Omron Sysmac Studio project Cobot_Test_200521 (Sysmac Studio 1.40.0.64008, StandardProject)

# Controller new_Controller_0: NX102-9020 version 1.34
Units and slaves: Unit 1 : NX-PF0730 (N2); Unit 2 : NX-AD3203 (N3); Unit 3 : NX-ID5442 (N4); Unit 4 : NX-OC4633 (N1); Unit 5 : NX-OC4633 (N7)
Task PrimaryTask (priority 4, period or condition 2000): Main, TM_Movements_Connection, TM_Movements, CobotModbusComms
Library TM_Commands 1.2.1 (contents left out)
Library TMmodbus Lib FW1.80 FB3.0.03 3.0.03 (contents left out)

TYPE PointStruct : STRUCT
    PosX : REAL;
    PosY : REAL;
    PosZ : REAL;
    PosRx : REAL;
    PosRy : REAL;
    PosRz : REAL;
END_STRUCT END_TYPE
TYPE PointStruct_STR : STRUCT
    PosX : STRING[10];
    PosY : STRING[10];
    PosZ : STRING[10];
    PosRx : STRING[10];
    PosRy : STRING[10];
    PosRz : STRING[10];
END_STRUCT END_TYPE
TYPE RobPosDK : STRUCT  (* TM12 move cmd from RoboDK *)
    MovType : STRING[15];  (* Move Type (PTP,Line,Circle) *)
    RobPosX : REAL;  (* X axis coordinates *)
    RobPosY : REAL;  (* Y axis coordinates *)
    RobPosZ : REAL;  (* Z axis coordinates *)
    RobPosRx : REAL;  (* Rotational X axis coordinates *)
    RobPosRy : REAL;  (* Rotational Y axis coordinates *)
    RobPosRz : REAL;  (* Rotational Z axis coordinates *)
    VarIO : STRING[20];
END_STRUCT END_TYPE
TYPE JobStruct : STRUCT
    JobID : INT;
    PartID : STRING[50];
    Qty : INT;
    EstTime : STRING[50];
    StartTimeDate : STRING[50];
    JobType : STRING[50];
    TimeAdded : DATE_AND_TIME;
END_STRUCT END_TYPE

VAR_GLOBAL RETAIN
    StartCommunications : BOOL;  (* published *)
END_VAR
VAR_GLOBAL
    MBerror : WORD;  (* published *)
    RobotCoordinates : TMmodbus\sRobotCoordinate;  (* published *)
    TouchCoordinates : TMmodbus\sRobotCoordinateTouch;  (* published *)
    RobotStatus : TMmodbus\sRobotStatus;  (* published *)
    RobotVitals : TMmodbus\sRobotVitals;  (* published *)
    Config : TMmodbus\sConfiguration;  (* published *)
    RobotJointTorques : TMmodbus\sRobotJointTorque;  (* published *)
    RobotTCPLive : TMmodbus\sRobotTCPLive;  (* published *)
    CurrentProjectName : string[200];  (* published *)
    NewProjectName : string[200];  (* published *)
    CommsRoundRobin : REAL;  (* published *)
    TCPerror : WORD;  (* published *)
    RobotControlBoxInfo : TMmodbus\sRobotControllerData;  (* published *)
    Buttons : TMmodbus\sRobotStickButtons;  (* published *)
    RobotIO : TMmodbus\sRobotIO;  (* published *)
    RobotSafetySettings : TMmodbus\sRobotSafety;  (* published *)
    RealsToRobot : ARRAY[0..49] OF real;  (* published *)
    FloatsFromRobot : ARRAY[0..49] OF real;  (* published *)
    BoolsToRobot : ARRAY[0..63] OF BOOL;  (* published *)
    Int16sFromRobot : ARRAY[0..49] OF INT;  (* published *)
    BoolsFromRobot : ARRAY[0..63] OF BOOL;  (* published *)
    IntsToRobot : ARRAY[0..49] OF INT;  (* published *)
    CommunicationsStatus : _eCONNECTION_STATE;  (* published *)
    CommunicationsBusy : BOOL;  (* published *)
    TCPerrorOriginator : TMModbus\eFunctionBlockError;  (* published *)
    RetryCounter : UINT;  (* published *)
    Stitching_Status : DINT;  (* published *)
    Stitching_Speed : REAL;  (* published *)
    Robot_Status : DINT;  (* published *)
    RobPos_X : DINT;  (* published *)
    RobPos_Y : DINT;  (* published *)
    RobPos_Z : DINT;  (* published *)
    Relay_Output : BYTE;  (* at IOBus://unit#4/Output Bit 8 bits; published *)
    Relay_Output1 : BOOL;  (* at IOBus://unit#4/Output Bit 8 bits/Output Bit 00; published *)
    Relay_Output2 : BOOL;  (* at IOBus://unit#4/Output Bit 8 bits/Output Bit 01; published *)
    Relay_Output3 : BOOL;  (* at IOBus://unit#4/Output Bit 8 bits/Output Bit 02; published *)
    Relay_Output4 : BOOL;  (* at IOBus://unit#4/Output Bit 8 bits/Output Bit 03; published *)
    Run_Stiching : BOOL;  (* published *)
    StartProgram : BOOL;  (* published *)
    CableConnected : BOOL;  (* published *)
    MTCP_Connect_TCP_Socket : _sSOCKET;  (* published *)
    MTCP_Connect_Connected : BOOL;
    ListenNode_Connect_Connected : BOOL;
    ListenNode_Connect_TCP_Socket : _sSOCKET;
    TaskTimeFB : REAL;
    Speed : REAL;  (* published *)
    TM_ReadPosition_X : REAL;
    TM_ReadPosition_Y : REAL;
    TM_ReadPosition_Z : REAL;  (* published *)
    Register : ARRAY[0..1023] OF WORD;
    TM_MovCmd_Command : STRING[256];
    Stitching_InManual : BOOL;
    Vision_IN : ARRAY[0..495] OF BYTE;  (* network input *)
    Vision_OUT : ARRAY[0..495] OF BYTE;  (* network output *)
    Part_Orientation_DINT : DINT;
    Part_Dist_X : DINT;
    Part_Dist_Y : DINT;
    Vision_Result_OK : DINT;  (* published *)
    Part_Orientation_REAL : REAL;
    Rz_Attach : REAL;
    RZ_Attach_String : STRING[256] := '';
    X_Attach_String : String[10];
    Y_Attach_String : STRING[10];
END_VAR
VAR_GLOBAL RETAIN
    AttachPoint : PointStruct;
END_VAR
VAR_GLOBAL
    AttachPoint_STR : PointStruct_STR;
    Z_Attach_String : string[10];
    Rx_Attach_String : string[10];
    Ry_Attach_String : string[10];
    Attach : STRING[256];
    RobPosTM : ARRAY[0..100] OF RobPosDK;
    CSVstrings : ARRAY[0..100] OF STRING[100];
    Position_STR : ARRAY[0..100] OF PointStruct_STR;
    Position1 : STRING[256];
    Position : ARRAY[0..100] OF STRING[100];
    MovType : ARRAY[0..100] OF STRING[100];
    RoboDKLoad : BOOL;  (* published *)
    FileName : STRING[100];  (* published *)
    ProgramToLoad : STRING[100];
    Index_STR : DINT;
    AI_CH1 : INT;  (* at IOBus://unit#2/Ch1 Analog Input Value; published *)
    AI_CH2 : INT;  (* at IOBus://unit#2/Ch2 Analog Input Value; published *)
    AI_CH3 : INT;  (* at IOBus://unit#2/Ch3 Analog Input Value; published *)
    AI_CH4 : INT;  (* at IOBus://unit#2/Ch4 Analog Input Value; published *)
    N4_Input_Bit_00 : BOOL;  (* at IOBus://unit#3/Input Bit 16 bits/Input Bit 00 *)
    N4_Input_Bit_01 : BOOL;  (* at IOBus://unit#3/Input Bit 16 bits/Input Bit 01 *)
    N4_Input_Bit_02 : BOOL;  (* at IOBus://unit#3/Input Bit 16 bits/Input Bit 02 *)
    N4_Input_Bit_03 : BOOL;  (* at IOBus://unit#3/Input Bit 16 bits/Input Bit 03 *)
    N4_Input_Bit_04 : BOOL;  (* at IOBus://unit#3/Input Bit 16 bits/Input Bit 04 *)
    N4_Input_Bit_05 : BOOL;  (* at IOBus://unit#3/Input Bit 16 bits/Input Bit 05 *)
    DistanceSensor : REAL;
    Relay_Output5 : BOOL;  (* at IOBus://unit#4/Output Bit 8 bits/Output Bit 04 *)
    Relay_Output6 : BOOL;  (* at IOBus://unit#4/Output Bit 8 bits/Output Bit 05 *)
    Relay_Output7 : BOOL;  (* at IOBus://unit#4/Output Bit 8 bits/Output Bit 06 *)
    Relay_Output8 : BOOL;  (* at IOBus://unit#4/Output Bit 8 bits/Output Bit 07 *)
    Bottom_Cyl_IN : BOOL;
    Bottom_Cyl_OUT : BOOL;
    Striker_Plt_DOWN : BOOL;
    Striker_Plt_UP : BOOL;
    Cutter_IN : BOOL;
    Cutter_OUT : BOOL;
    Top_N_Bottom_Cut_D : BOOL;
    Striker_Plate_D : BOOL;
    Vacuum_D : BOOL;
    Main_Cut_D : BOOL;
    Alarms_Int : DINT;  (* published *)
    Rob_Speed : DINT;  (* published *)
    GRAFANA_Counter : INT;  (* published *)
    Taping_Status : DINT;  (* published *)
    Run_Taping : BOOL;
END_VAR
VAR_GLOBAL RETAIN
    Parts_06Hrs : DINT;  (* published *)
    Parts_07Hrs : DINT;  (* published *)
    Parts_08Hrs : DINT;  (* published *)
    Parts_09Hrs : DINT;  (* published *)
    Parts_10Hrs : DINT;  (* published *)
    Parts_11Hrs : DINT;  (* published *)
    Parts_12Hrs : DINT;  (* published *)
    Parts_13Hrs : DINT;  (* published *)
    Parts_14Hrs : DINT;  (* published *)
    Parts_15Hrs : DINT;  (* published *)
    Parts_16Hrs : DINT;  (* published *)
    Parts_17Hrs : DINT;  (* published *)
    Parts_SP : DINT;  (* published *)
END_VAR
VAR_GLOBAL
    Stitching_OEE : DINT;  (* published *)
    Taping_OEE : DINT;  (* published *)
    RobProgIO : ARRAY[0..100] OF STRING[25];
    Run_Stiching_Man : BOOL;  (* published *)
    Stitcher_AutoSpeed : BOOL;
    Proj_Rob_Speed : INT;
    VarIO : ARRAY[0..100] OF STRING[100];
    Relay_Output9 : BOOL;  (* at IOBus://unit#5/Output Bit 8 bits/Output Bit 00 *)
    ERPJob : JobStruct;  (* published *)
    ERPJobWorking : JobStruct;
END_VAR
VAR_GLOBAL CONSTANT
    ERPJobZero : JobStruct;
END_VAR

PROGRAM Main
VAR
    Input1 : BOOL;  (* Enter Variable Commen *)
    Input2 : BOOL;
    Input3 : BOOL;
    Input4 : BOOL;
    RobotPos_Stiching : BOOL;
    xPlaceholder : DINT;
    yPlaceholder : DINT;
    zPlaceholder : DINT;
    placeholder : BOOL;
    Robot_Running : BOOL;
    Rb_Error_Present : BOOL;
    St_Error_Present : BOOL;
    CommunicationsBusy : BOOL;
    StartCommunications : BOOL;
    Start : BOOL;
    def : BOOL;
    testt : BOOL;
    X_Attach : REAL;
    Y_Attach : REAL;
    Part_Dist_X_REAL : REAL;
    Part_Dist_Y_REAL : REAL;
    X_temp : REAL;
    Y_temp : REAL;
    TrigRoboProgramRead : BOOL;
    OpenRoboProgram : FileOpen;
    OpenFileError : BOOL;
    ProgramToOpen : STRING[255];
    Fid : DWORD;
    ReadRoboProgram : FileGets;
    ReadFileError : BOOL;
    Index : DINT;
    CloseRoboProgram : FileClose;
    CloseFileError : BOOL;
    ReadComplete : BOOL;
    OperatingEnd : BOOL;
    Trigger : BOOL;
    RS_Instance : RS;
    tuti : BOOL;
    OpenProgramName : STRING[100];
    x : BOOL;
    i : DINT;
    R_TRIG_instance : R_TRIG;
    Stp : DINT;
    Vis_Error_Present : BOOL;
    Rob_Alarm : BOOL;
    St_Alarm : BOOL;
    Vis_Alarm : BOOL;
    GRAFANA_TON : TON;
    GRAFANA_TON_ET : TIME;
    GRAFANA_CTU : CTU;
    Reset_Counter : BOOL;
    Tp_Error_Present : BOOL;
    Tp_Alarm : BOOL;
    Speed_mms : DINT;
    StepMove : DINT;
    temp : UINT;
    Load : BOOL;
    LoadSchedule : BOOL;
    ScheduleName : STRING[100];
    TrigScheduleRead : BOOL;
    OpenSchedule : FileOpen;
    ReadSchedule : FileGets;
    CloseSchedule : FileClose;
    BackStitch_TON : TON;
    BackStitch_TON_ACC : TIME;
    MoveERPData : BOOL;
    abc : _sTimer;
    timeret : UINT;
    q : BOOL;
    TON12 : TON;
    afd : TIME;
    tesss : BOOL;
    ClearERPData : BOOL;
END_VAR
VAR_EXTERNAL
    Stitching_Status : DINT;
    Stitching_Speed : REAL;
    Robot_Status : DINT;
    Relay_Output : BYTE;
    RobPos_X : DINT;
    RobPos_Y : DINT;
    RobPos_Z : DINT;
    RobotCoordinates : TMmodbus\sRobotCoordinate;
    RobotStatus : TMmodbus\sRobotStatus;
    Run_Stiching : BOOL;
    Speed : REAL;
    Vision_IN : ARRAY[0..495] OF BYTE;
    Part_Orientation_DINT : DINT;
    Part_Dist_X : DINT;
    Part_Dist_Y : DINT;
    Vision_OUT : ARRAY[0..495] OF BYTE;
    Part_Orientation_REAL : REAL;
    Rz_Attach : REAL;
    RZ_Attach_String : STRING[256];
    X_Attach_String : String[10];
    Y_Attach_String : STRING[10];
    AttachPoint : PointStruct;
    Z_Attach_String : string[10];
    RX_Attach_String : string[10];
    RY_Attach_String : string[10];
    AttachPoint_STR : PointStruct_STR;
    Attach : STRING[256];
    Vision_Result_OK : DINT;
END_VAR
VAR_EXTERNAL CONSTANT
    _Card1Ready : BOOL;
END_VAR
VAR_EXTERNAL
    RobPosTM : ARRAY[0..100] OF RobPosDK;
    CSVstrings : ARRAY[0..100] OF STRING[100];
    Position1 : STRING[256];
    Position_STR : ARRAY[0..100] OF PointStruct_STR;
    Position : ARRAY[0..100] OF STRING[100];
    MovType : ARRAY[0..100] OF STRING[100];
    RoboDKLoad : BOOL;
    FileName : STRING[100];
    Index_STR : DINT;
    AI_CH1 : INT;
    DistanceSensor : REAL;
    N4_Input_Bit_00 : BOOL;
    N4_Input_Bit_01 : BOOL;
    N4_Input_Bit_02 : BOOL;
    N4_Input_Bit_03 : BOOL;
    N4_Input_Bit_04 : BOOL;
    N4_Input_Bit_05 : BOOL;
    Relay_Output5 : BOOL;
    Relay_Output6 : BOOL;
    Relay_Output7 : BOOL;
    Bottom_Cyl_IN : BOOL;
    Bottom_Cyl_OUT : BOOL;
    Striker_Plt_DOWN : BOOL;
    Striker_Plt_UP : BOOL;
    Cutter_IN : BOOL;
    Cutter_OUT : BOOL;
    Top_N_Bottom_Cut_D : BOOL;
    Striker_Plate_D : BOOL;
    Vacuum_D : BOOL;
    Relay_Output8 : BOOL;
    Main_Cut_D : BOOL;
    ListenNode_Connect_Connected : BOOL;
    Alarms_Int : DINT;
    RobotTCPLive : TMmodbus\sRobotTCPLive;
    Rob_Speed : DINT;
    GRAFANA_Counter : INT;
    Taping_Status : DINT;
    Run_Taping : BOOL;
    RobProgIO : ARRAY[0..100] OF STRING[25];
    Run_Stiching_Man : BOOL;
    Stitcher_AutoSpeed : BOOL;
    StartProgram : BOOL;
    VarIO : ARRAY[0..100] OF STRING[100];
    Relay_Output9 : BOOL;
    ERPJob : JobStruct;
    ERPJobWorking : JobStruct;
END_VAR
VAR_EXTERNAL CONSTANT
    ERPJobZero : JobStruct;
END_VAR
VAR
    _e1 : R_TRIG;
    _p2 : BOOL;
    _p3 : BOOL;
    _p4 : BOOL;
    _p5 : BOOL;
    _p6 : BOOL;
    _p7 : BOOL;
    _p8 : BOOL;
    _p9 : BOOL;
    _p10 : BOOL;
    _p11 : BOOL;
    _p12 : BOOL;
    _p13 : BOOL;
    _p14 : BOOL;
    _p15 : BOOL;
    _p16 : BOOL;
    _e17 : F_TRIG;
    _e18 : F_TRIG;
    _e19 : R_TRIG;
    _e20 : R_TRIG;
    _e21 : R_TRIG;
    _p22 : BOOL;
    _p23 : BOOL;
    _e24 : R_TRIG;
    _e25 : R_TRIG;
END_VAR

(* Section DataToGrafana: ladder, written here as Structured Text *)

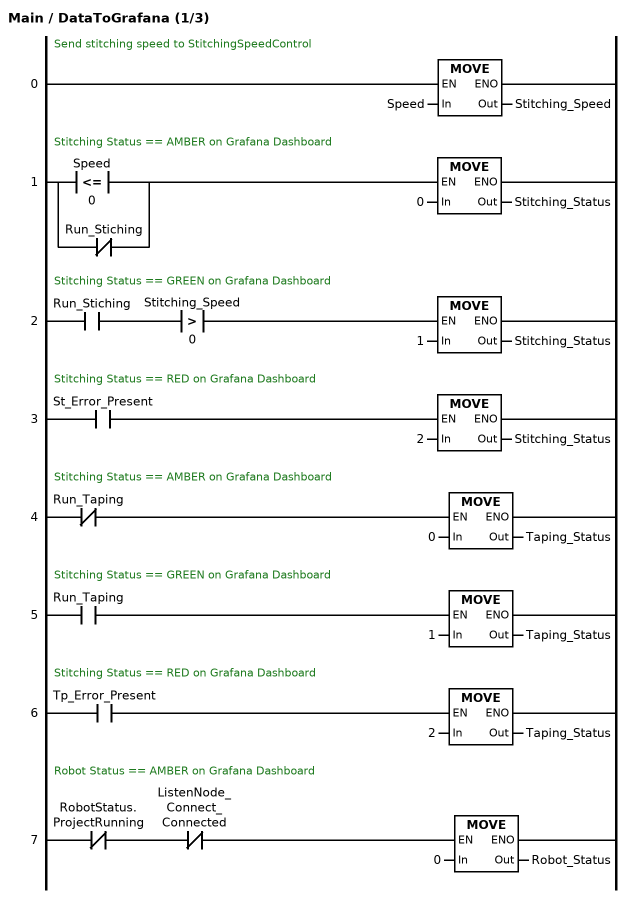
(* Rung 0: Send stitching speed to StitchingSpeedControl *)
Stitching_Speed := Speed;
(* Rung 1: Stitching Status == AMBER on Grafana Dashboard *)
IF (Speed <= 0) OR NOT Run_Stiching THEN Stitching_Status := 0; END_IF;
(* Rung 2: Stitching Status == GREEN on Grafana Dashboard *)
IF Run_Stiching AND (Stitching_Speed > 0) THEN Stitching_Status := 1; END_IF;
(* Rung 3: Stitching Status == RED on Grafana Dashboard *)
IF St_Error_Present THEN Stitching_Status := 2; END_IF;
(* Rung 4: Stitching Status == AMBER on Grafana Dashboard *)
IF NOT Run_Taping THEN Taping_Status := 0; END_IF;
(* Rung 5: Stitching Status == GREEN on Grafana Dashboard *)
IF Run_Taping THEN Taping_Status := 1; END_IF;
(* Rung 6: Stitching Status == RED on Grafana Dashboard *)
IF Tp_Error_Present THEN Taping_Status := 2; END_IF;
(* Rung 7: Robot Status == AMBER on Grafana Dashboard *)
IF NOT RobotStatus.ProjectRunning AND NOT ListenNode_Connect_Connected THEN Robot_Status := 0; END_IF;

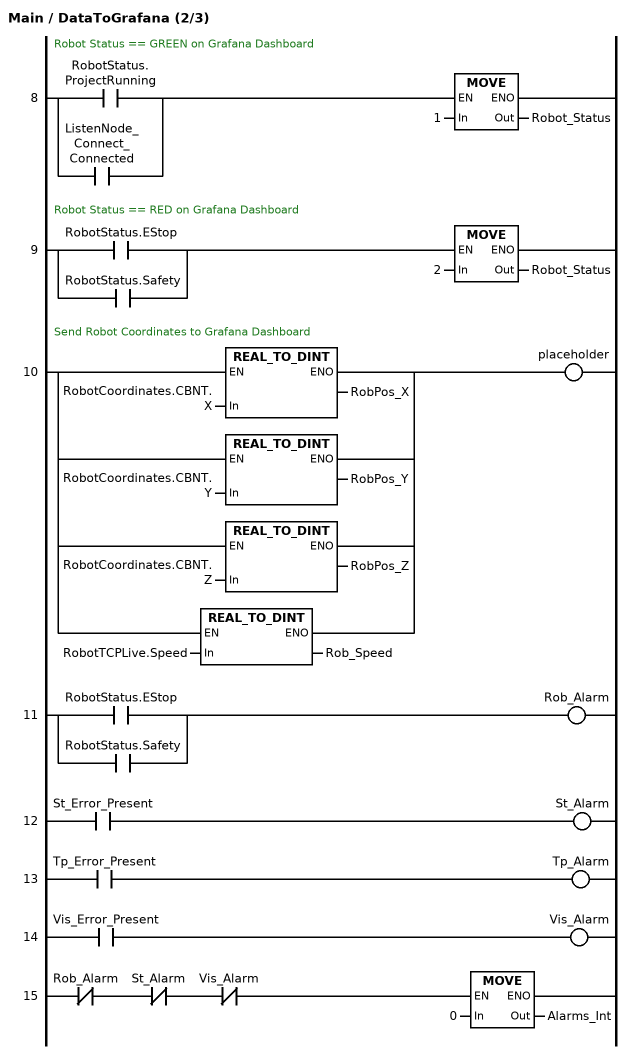
(* Rung 8: Robot Status == GREEN on Grafana Dashboard *)
IF RobotStatus.ProjectRunning OR ListenNode_Connect_Connected THEN Robot_Status := 1; END_IF;
(* Rung 9: Robot Status == RED on Grafana Dashboard *)
IF RobotStatus.EStop OR RobotStatus.Safety THEN Robot_Status := 2; END_IF;
(* Rung 10: Send Robot Coordinates to Grafana Dashboard *)
RobPos_X := REAL_TO_DINT(In := RobotCoordinates.CBNT.X);
RobPos_Y := REAL_TO_DINT(In := RobotCoordinates.CBNT.Y);
RobPos_Z := REAL_TO_DINT(In := RobotCoordinates.CBNT.Z);
Rob_Speed := REAL_TO_DINT(In := RobotTCPLive.Speed);
placeholder := TRUE;
(* Rung 11 *)
Rob_Alarm := RobotStatus.EStop OR RobotStatus.Safety;
(* Rung 12 *)
St_Alarm := St_Error_Present;
(* Rung 13 *)
Tp_Alarm := Tp_Error_Present;
(* Rung 14 *)
Vis_Alarm := Vis_Error_Present;
(* Rung 15 *)
IF NOT Rob_Alarm AND NOT St_Alarm AND NOT Vis_Alarm THEN Alarms_Int := 0; END_IF;

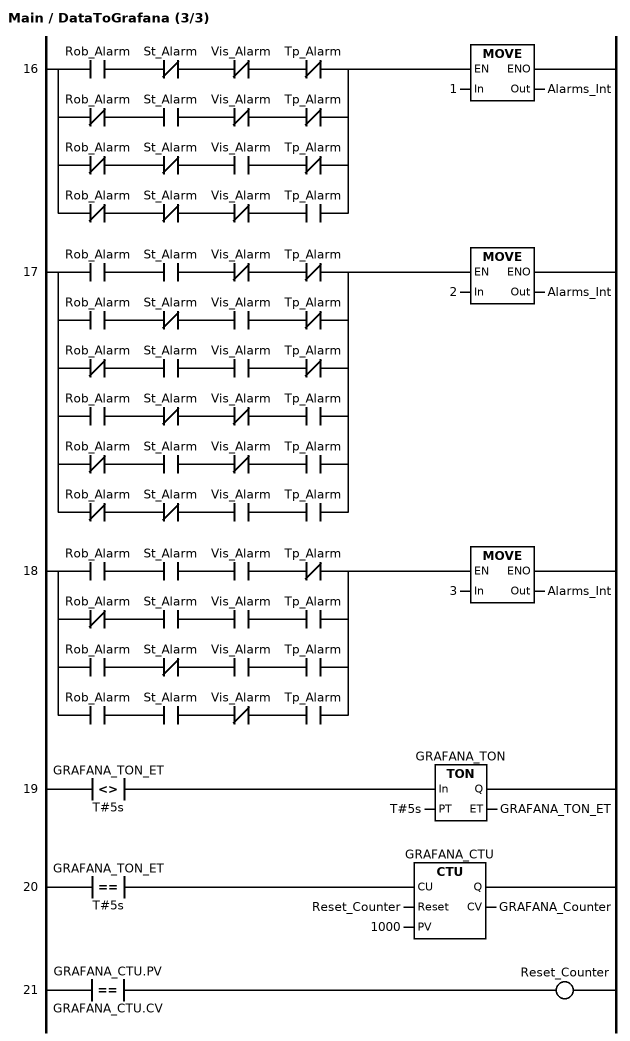
(* Rung 16 *)
IF (Rob_Alarm AND NOT St_Alarm AND NOT Vis_Alarm AND NOT Tp_Alarm) OR (NOT Rob_Alarm AND St_Alarm AND NOT Vis_Alarm AND NOT Tp_Alarm) OR (NOT Rob_Alarm AND NOT St_Alarm AND Vis_Alarm AND NOT Tp_Alarm) OR (NOT Rob_Alarm AND NOT St_Alarm AND NOT Vis_Alarm AND Tp_Alarm) THEN
    Alarms_Int := 1;
END_IF;
(* Rung 17 *)
IF (Rob_Alarm AND St_Alarm AND NOT Vis_Alarm AND NOT Tp_Alarm) OR (Rob_Alarm AND NOT St_Alarm AND Vis_Alarm AND NOT Tp_Alarm) OR (NOT Rob_Alarm AND St_Alarm AND Vis_Alarm AND NOT Tp_Alarm) OR (Rob_Alarm AND NOT St_Alarm AND NOT Vis_Alarm AND Tp_Alarm) OR (NOT Rob_Alarm AND St_Alarm AND NOT Vis_Alarm AND Tp_Alarm) OR (NOT Rob_Alarm AND NOT St_Alarm AND Vis_Alarm AND Tp_Alarm) THEN
    Alarms_Int := 2;
END_IF;
(* Rung 18 *)
IF (Rob_Alarm AND St_Alarm AND Vis_Alarm AND NOT Tp_Alarm) OR (NOT Rob_Alarm AND St_Alarm AND Vis_Alarm AND Tp_Alarm) OR (Rob_Alarm AND NOT St_Alarm AND Vis_Alarm AND Tp_Alarm) OR (Rob_Alarm AND St_Alarm AND NOT Vis_Alarm AND Tp_Alarm) THEN
    Alarms_Int := 3;
END_IF;
(* Rung 19 *)
GRAFANA_TON(In := GRAFANA_TON_ET <> T#5s, PT := T#5s, ET => GRAFANA_TON_ET);
(* Rung 20 *)
_e1(CLK := GRAFANA_TON_ET = T#5s);
GRAFANA_CTU(CU := _e1.Q, Reset := Reset_Counter, PV := 1000, CV => GRAFANA_Counter);
(* Rung 21 *)
Reset_Counter := GRAFANA_CTU.PV = GRAFANA_CTU.CV;

(* Section StichingMachine: ladder, written here as Structured Text *)

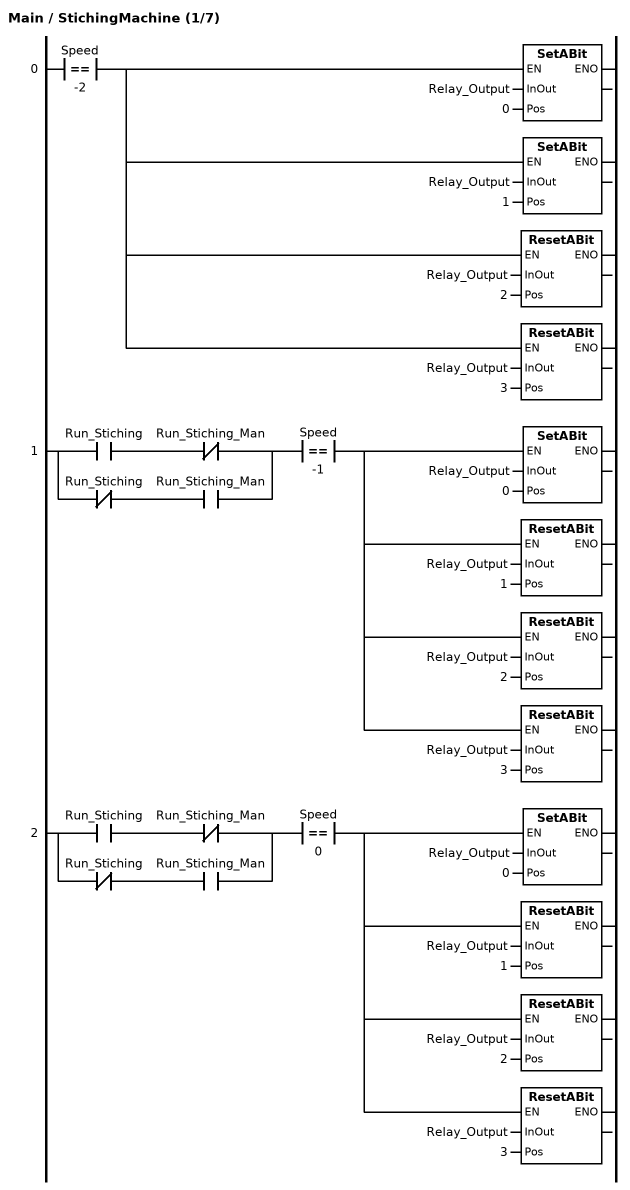
(* Rung 0 *)
IF Speed = -2 THEN
    SetABit(InOut := Relay_Output, Pos := 0);
    SetABit(InOut := Relay_Output, Pos := 1);
    ResetABit(InOut := Relay_Output, Pos := 2);
    ResetABit(InOut := Relay_Output, Pos := 3);
END_IF;
(* Rung 1 *)
_p2 := ((Run_Stiching AND NOT Run_Stiching_Man) OR (NOT Run_Stiching AND Run_Stiching_Man)) AND (Speed = -1);
IF _p2 THEN
    SetABit(InOut := Relay_Output, Pos := 0);
    ResetABit(InOut := Relay_Output, Pos := 1);
    ResetABit(InOut := Relay_Output, Pos := 2);
    ResetABit(InOut := Relay_Output, Pos := 3);
END_IF;
(* Rung 2 *)
_p3 := ((Run_Stiching AND NOT Run_Stiching_Man) OR (NOT Run_Stiching AND Run_Stiching_Man)) AND (Speed = 0);
IF _p3 THEN
    SetABit(InOut := Relay_Output, Pos := 0);
    ResetABit(InOut := Relay_Output, Pos := 1);
    ResetABit(InOut := Relay_Output, Pos := 2);
    ResetABit(InOut := Relay_Output, Pos := 3);
END_IF;

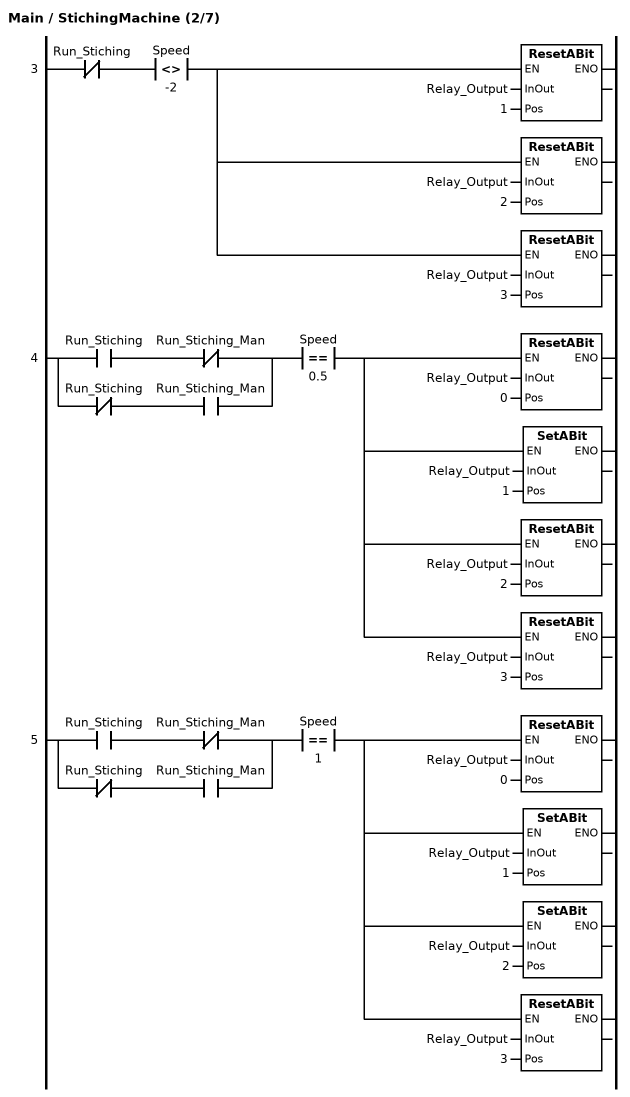
(* Rung 3 *)
IF NOT Run_Stiching AND (Speed <> -2) THEN
    ResetABit(InOut := Relay_Output, Pos := 1);
    ResetABit(InOut := Relay_Output, Pos := 2);
    ResetABit(InOut := Relay_Output, Pos := 3);
END_IF;
(* Rung 4 *)
_p4 := ((Run_Stiching AND NOT Run_Stiching_Man) OR (NOT Run_Stiching AND Run_Stiching_Man)) AND (Speed = 0.5);
IF _p4 THEN
    ResetABit(InOut := Relay_Output, Pos := 0);
    SetABit(InOut := Relay_Output, Pos := 1);
    ResetABit(InOut := Relay_Output, Pos := 2);
    ResetABit(InOut := Relay_Output, Pos := 3);
END_IF;
(* Rung 5 *)
_p5 := ((Run_Stiching AND NOT Run_Stiching_Man) OR (NOT Run_Stiching AND Run_Stiching_Man)) AND (Speed = 1);
IF _p5 THEN
    ResetABit(InOut := Relay_Output, Pos := 0);
    SetABit(InOut := Relay_Output, Pos := 1);
    SetABit(InOut := Relay_Output, Pos := 2);
    ResetABit(InOut := Relay_Output, Pos := 3);
END_IF;

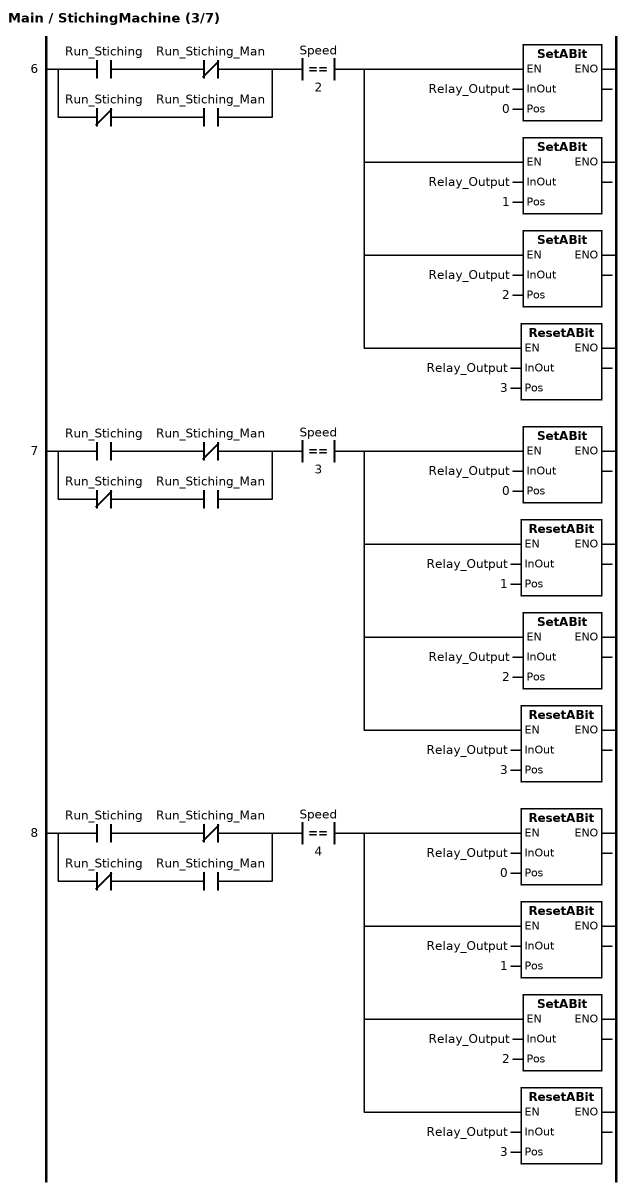
(* Rung 6 *)
_p6 := ((Run_Stiching AND NOT Run_Stiching_Man) OR (NOT Run_Stiching AND Run_Stiching_Man)) AND (Speed = 2);
IF _p6 THEN
    SetABit(InOut := Relay_Output, Pos := 0);
    SetABit(InOut := Relay_Output, Pos := 1);
    SetABit(InOut := Relay_Output, Pos := 2);
    ResetABit(InOut := Relay_Output, Pos := 3);
END_IF;
(* Rung 7 *)
_p7 := ((Run_Stiching AND NOT Run_Stiching_Man) OR (NOT Run_Stiching AND Run_Stiching_Man)) AND (Speed = 3);
IF _p7 THEN
    SetABit(InOut := Relay_Output, Pos := 0);
    ResetABit(InOut := Relay_Output, Pos := 1);
    SetABit(InOut := Relay_Output, Pos := 2);
    ResetABit(InOut := Relay_Output, Pos := 3);
END_IF;
(* Rung 8 *)
_p8 := ((Run_Stiching AND NOT Run_Stiching_Man) OR (NOT Run_Stiching AND Run_Stiching_Man)) AND (Speed = 4);
IF _p8 THEN
    ResetABit(InOut := Relay_Output, Pos := 0);
    ResetABit(InOut := Relay_Output, Pos := 1);
    SetABit(InOut := Relay_Output, Pos := 2);
    ResetABit(InOut := Relay_Output, Pos := 3);
END_IF;

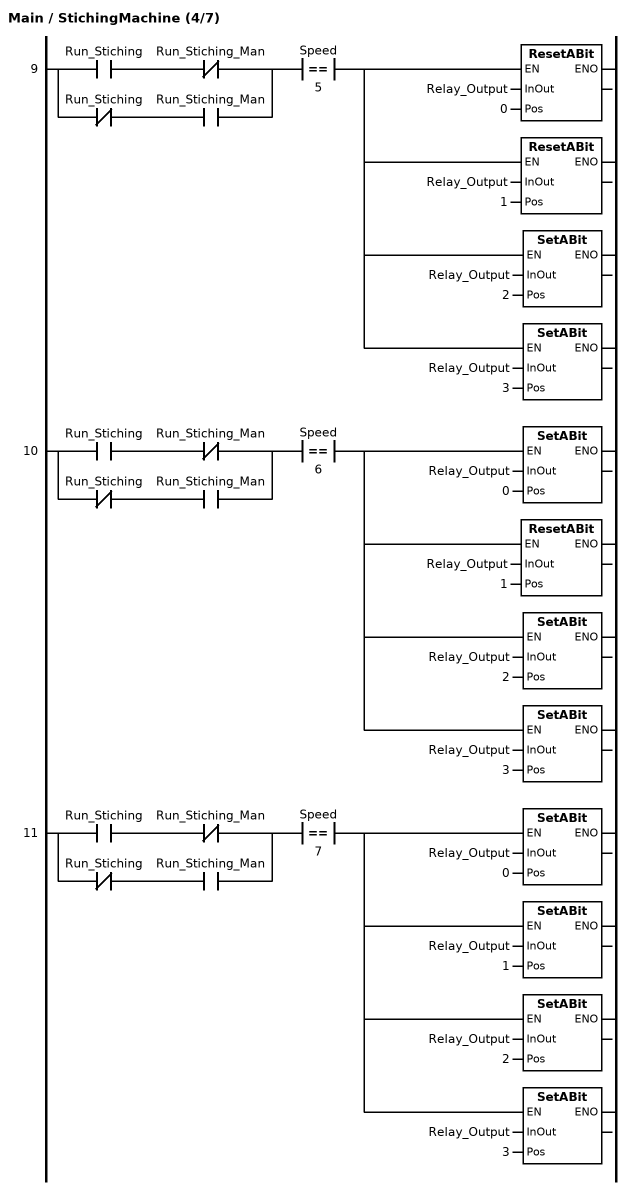
(* Rung 9 *)
_p9 := ((Run_Stiching AND NOT Run_Stiching_Man) OR (NOT Run_Stiching AND Run_Stiching_Man)) AND (Speed = 5);
IF _p9 THEN
    ResetABit(InOut := Relay_Output, Pos := 0);
    ResetABit(InOut := Relay_Output, Pos := 1);
    SetABit(InOut := Relay_Output, Pos := 2);
    SetABit(InOut := Relay_Output, Pos := 3);
END_IF;
(* Rung 10 *)
_p10 := ((Run_Stiching AND NOT Run_Stiching_Man) OR (NOT Run_Stiching AND Run_Stiching_Man)) AND (Speed = 6);
IF _p10 THEN
    SetABit(InOut := Relay_Output, Pos := 0);
    ResetABit(InOut := Relay_Output, Pos := 1);
    SetABit(InOut := Relay_Output, Pos := 2);
    SetABit(InOut := Relay_Output, Pos := 3);
END_IF;
(* Rung 11 *)
_p11 := ((Run_Stiching AND NOT Run_Stiching_Man) OR (NOT Run_Stiching AND Run_Stiching_Man)) AND (Speed = 7);
IF _p11 THEN
    SetABit(InOut := Relay_Output, Pos := 0);
    SetABit(InOut := Relay_Output, Pos := 1);
    SetABit(InOut := Relay_Output, Pos := 2);
    SetABit(InOut := Relay_Output, Pos := 3);
END_IF;

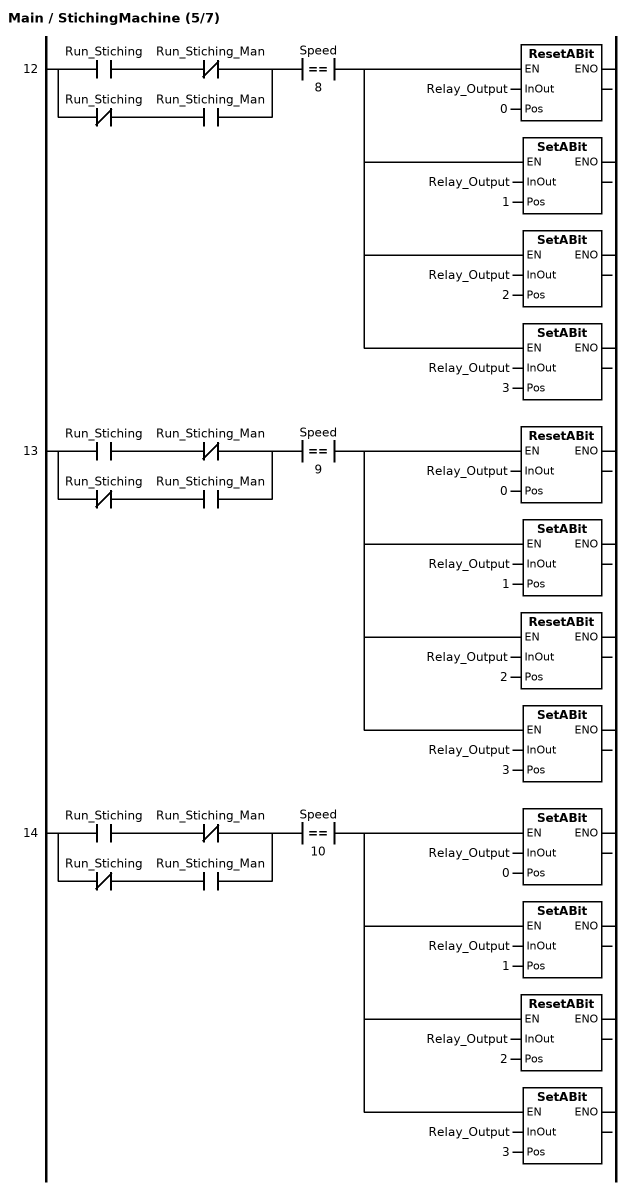
(* Rung 12 *)
_p12 := ((Run_Stiching AND NOT Run_Stiching_Man) OR (NOT Run_Stiching AND Run_Stiching_Man)) AND (Speed = 8);
IF _p12 THEN
    ResetABit(InOut := Relay_Output, Pos := 0);
    SetABit(InOut := Relay_Output, Pos := 1);
    SetABit(InOut := Relay_Output, Pos := 2);
    SetABit(InOut := Relay_Output, Pos := 3);
END_IF;
(* Rung 13 *)
_p13 := ((Run_Stiching AND NOT Run_Stiching_Man) OR (NOT Run_Stiching AND Run_Stiching_Man)) AND (Speed = 9);
IF _p13 THEN
    ResetABit(InOut := Relay_Output, Pos := 0);
    SetABit(InOut := Relay_Output, Pos := 1);
    ResetABit(InOut := Relay_Output, Pos := 2);
    SetABit(InOut := Relay_Output, Pos := 3);
END_IF;
(* Rung 14 *)
_p14 := ((Run_Stiching AND NOT Run_Stiching_Man) OR (NOT Run_Stiching AND Run_Stiching_Man)) AND (Speed = 10);
IF _p14 THEN
    SetABit(InOut := Relay_Output, Pos := 0);
    SetABit(InOut := Relay_Output, Pos := 1);
    ResetABit(InOut := Relay_Output, Pos := 2);
    SetABit(InOut := Relay_Output, Pos := 3);
END_IF;

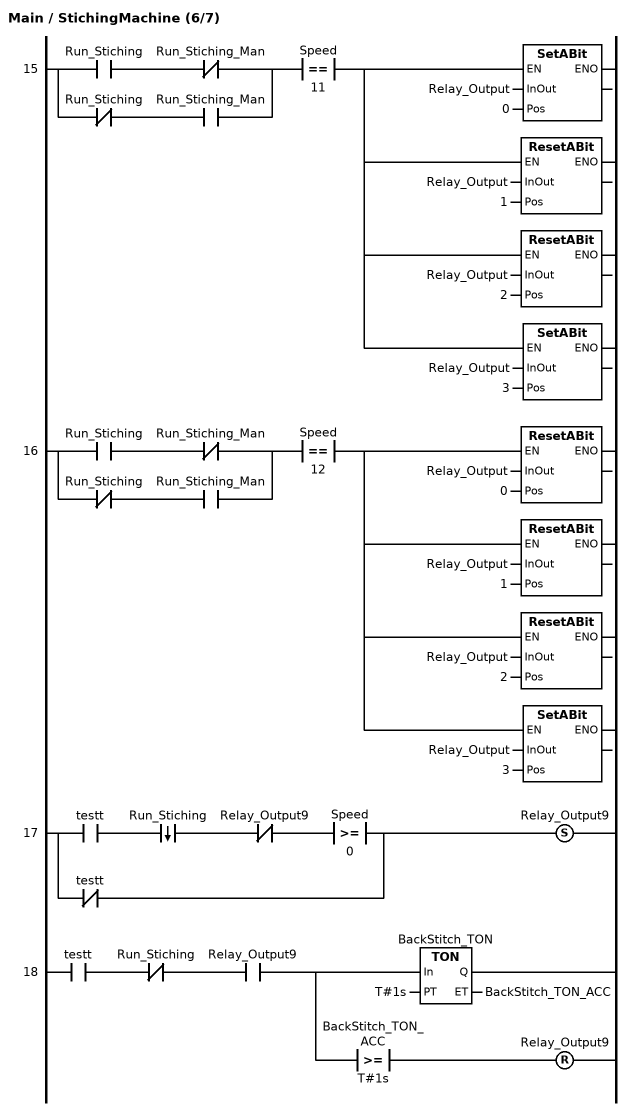
(* Rung 15 *)
_p15 := ((Run_Stiching AND NOT Run_Stiching_Man) OR (NOT Run_Stiching AND Run_Stiching_Man)) AND (Speed = 11);
IF _p15 THEN
    SetABit(InOut := Relay_Output, Pos := 0);
    ResetABit(InOut := Relay_Output, Pos := 1);
    ResetABit(InOut := Relay_Output, Pos := 2);
    SetABit(InOut := Relay_Output, Pos := 3);
END_IF;
(* Rung 16 *)
_p16 := ((Run_Stiching AND NOT Run_Stiching_Man) OR (NOT Run_Stiching AND Run_Stiching_Man)) AND (Speed = 12);
IF _p16 THEN
    ResetABit(InOut := Relay_Output, Pos := 0);
    ResetABit(InOut := Relay_Output, Pos := 1);
    ResetABit(InOut := Relay_Output, Pos := 2);
    SetABit(InOut := Relay_Output, Pos := 3);
END_IF;
(* Rung 17 *)
_e17(CLK := Run_Stiching);
IF (testt AND _e17.Q AND NOT Relay_Output9 AND (Speed >= 0)) OR NOT testt THEN
    Relay_Output9 := TRUE;
END_IF;
(* Rung 18 *)
BackStitch_TON(In := testt AND NOT Run_Stiching AND Relay_Output9, PT := T#1s, ET => BackStitch_TON_ACC);
IF testt AND NOT Run_Stiching AND Relay_Output9 AND (BackStitch_TON_ACC >= T#1s) THEN
    Relay_Output9 := FALSE;
END_IF;

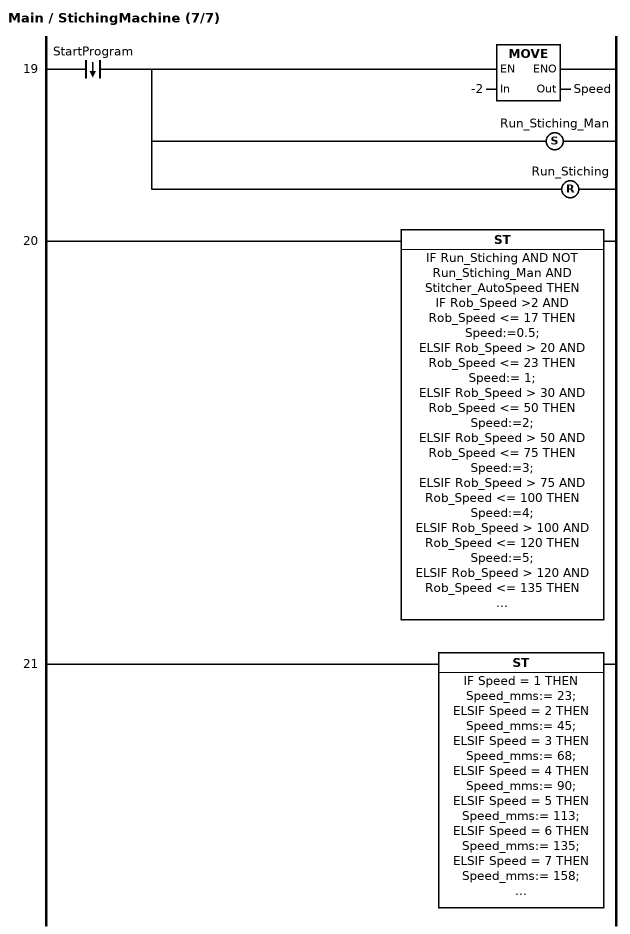
(* Rung 19 *)
_e18(CLK := StartProgram);
IF _e18.Q THEN
    Speed := -2;
    Run_Stiching_Man := TRUE;
    Run_Stiching := FALSE;
END_IF;
(* Rung 20 *)
IF Run_Stiching AND NOT Run_Stiching_Man AND Stitcher_AutoSpeed THEN
	IF Rob_Speed >2 AND Rob_Speed <= 17 THEN
		Speed:=0.5;
	ELSIF Rob_Speed > 20 AND Rob_Speed <= 23 THEN
		Speed:= 1; 
	ELSIF Rob_Speed > 30 AND Rob_Speed <= 50 THEN
		Speed:=2;
	 ELSIF Rob_Speed > 50 AND Rob_Speed <= 75 THEN
		Speed:=3;
	ELSIF Rob_Speed > 75 AND Rob_Speed <= 100 THEN
		Speed:=4;
	ELSIF Rob_Speed > 100 AND Rob_Speed <= 120 THEN
		Speed:=5;
	ELSIF Rob_Speed > 120 AND Rob_Speed <= 135 THEN
		Speed:=6;
	ELSIF Rob_Speed > 135 AND Rob_Speed <= 170 THEN
		Speed:=7;
	ELSIF Rob_Speed > 170 AND Rob_Speed <= 190 THEN
		Speed:=8;
	ELSIF Rob_Speed > 190 AND Rob_Speed <= 210 THEN
		Speed:=9;
	ELSIF Rob_Speed > 210 AND Rob_Speed <= 235 THEN
		Speed:=10;
	ELSIF Rob_Speed > 235 AND Rob_Speed <= 255 THEN
		Speed:=11;
	ELSIF Rob_Speed > 255 AND Rob_Speed <= 270 THEN
		Speed:=12;
	ELSIF Rob_Speed > 270 THEN
		Speed:=12;
	END_IF;
END_IF;
(* Rung 21 *)
IF Speed = 1 THEN
	Speed_mms:= 23;
ELSIF Speed = 2 THEN
	Speed_mms:= 45;
ELSIF Speed = 3 THEN
	Speed_mms:= 68;
ELSIF Speed = 4 THEN
	Speed_mms:= 90;
ELSIF Speed = 5 THEN
	Speed_mms:= 113;
ELSIF Speed = 6 THEN
	Speed_mms:= 135;	
ELSIF Speed = 7 THEN
	Speed_mms:= 158;
ELSIF Speed = 8 THEN
	Speed_mms:= 180;
ELSIF Speed = 9 THEN
	Speed_mms:= 203;
ELSIF Speed = 10 THEN
	Speed_mms:= 225;
ELSIF Speed = 11 THEN
	Speed_mms:= 248;
ELSIF Speed = 12 THEN
	Speed_mms:= 270;
END_IF;

(* Section VisionSystem: ladder, written here as Structured Text *)

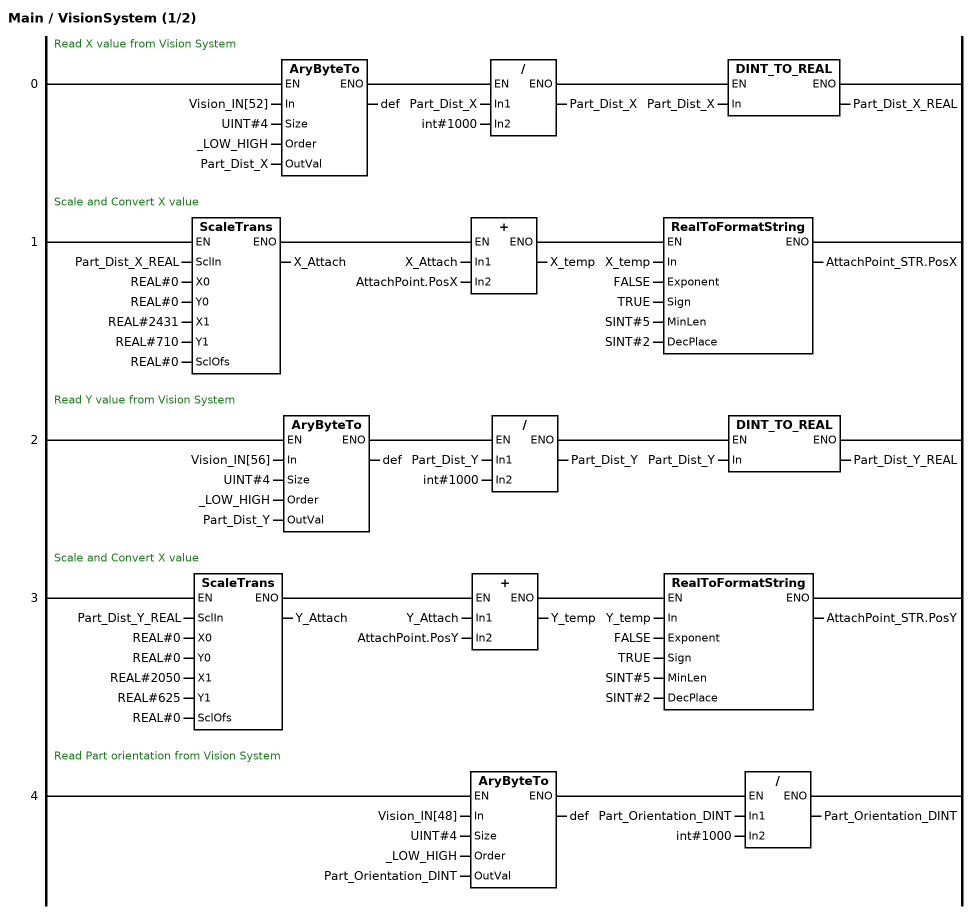
(* Rung 0: Read X value from Vision System *)
def := AryByteTo(In := Vision_IN[52], Size := UINT#4, Order := _LOW_HIGH, OutVal := Part_Dist_X);
Part_Dist_X := Part_Dist_X / int#1000;
Part_Dist_X_REAL := DINT_TO_REAL(In := Part_Dist_X);
(* Rung 1: Scale and Convert X value *)
X_Attach := ScaleTrans(SclIn := Part_Dist_X_REAL, X0 := REAL#0, Y0 := REAL#0, X1 := REAL#2431, Y1 := REAL#710, SclOfs := REAL#0);
X_temp := X_Attach + AttachPoint.PosX;
AttachPoint_STR.PosX := RealToFormatString(In := X_temp, Exponent := FALSE, Sign := TRUE, MinLen := SINT#5, DecPlace := SINT#2);
(* Rung 2: Read Y value from Vision System *)
def := AryByteTo(In := Vision_IN[56], Size := UINT#4, Order := _LOW_HIGH, OutVal := Part_Dist_Y);
Part_Dist_Y := Part_Dist_Y / int#1000;
Part_Dist_Y_REAL := DINT_TO_REAL(In := Part_Dist_Y);
(* Rung 3: Scale and Convert X value *)
Y_Attach := ScaleTrans(SclIn := Part_Dist_Y_REAL, X0 := REAL#0, Y0 := REAL#0, X1 := REAL#2050, Y1 := REAL#625, SclOfs := REAL#0);
Y_temp := Y_Attach + AttachPoint.PosY;
AttachPoint_STR.PosY := RealToFormatString(In := Y_temp, Exponent := FALSE, Sign := TRUE, MinLen := SINT#5, DecPlace := SINT#2);
(* Rung 4: Read Part orientation from Vision System *)
def := AryByteTo(In := Vision_IN[48], Size := UINT#4, Order := _LOW_HIGH, OutVal := Part_Orientation_DINT);
Part_Orientation_DINT := Part_Orientation_DINT / int#1000;

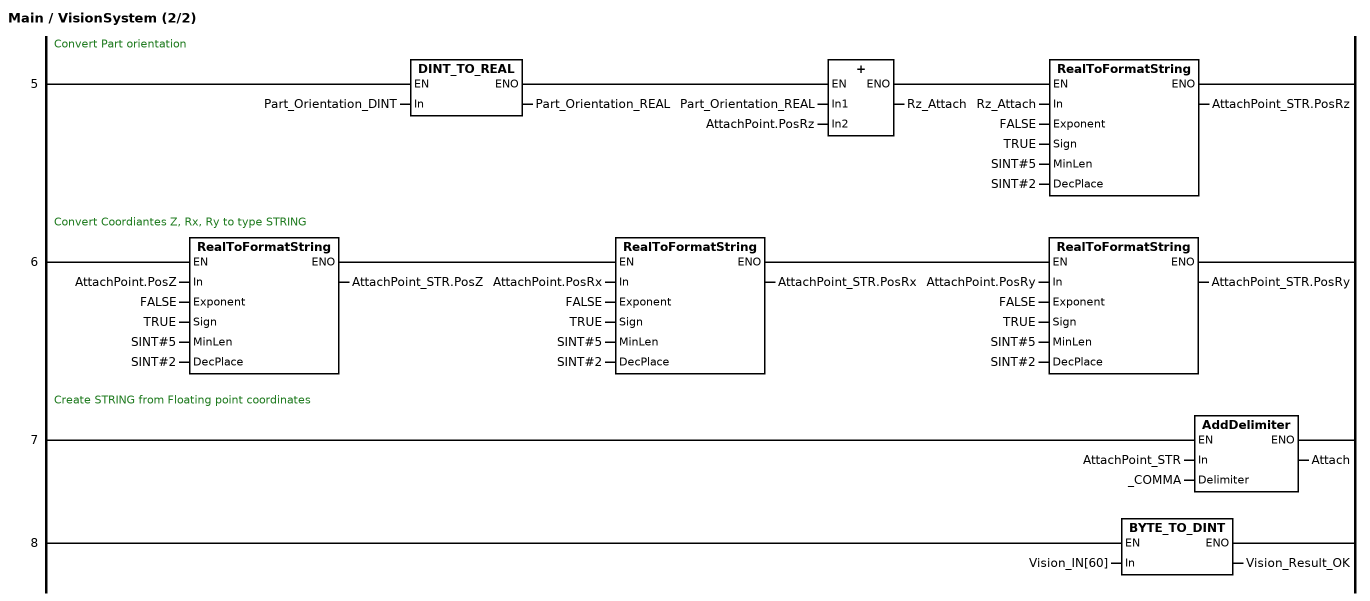
(* Rung 5: Convert Part orientation *)
Part_Orientation_REAL := DINT_TO_REAL(In := Part_Orientation_DINT);
Rz_Attach := Part_Orientation_REAL + AttachPoint.PosRz;
AttachPoint_STR.PosRz := RealToFormatString(In := Rz_Attach, Exponent := FALSE, Sign := TRUE, MinLen := SINT#5, DecPlace := SINT#2);
(* Rung 6: Convert Coordiantes Z, Rx, Ry to type STRING *)
AttachPoint_STR.PosZ := RealToFormatString(In := AttachPoint.PosZ, Exponent := FALSE, Sign := TRUE, MinLen := SINT#5, DecPlace := SINT#2);
AttachPoint_STR.PosRx := RealToFormatString(In := AttachPoint.PosRx, Exponent := FALSE, Sign := TRUE, MinLen := SINT#5, DecPlace := SINT#2);
AttachPoint_STR.PosRy := RealToFormatString(In := AttachPoint.PosRy, Exponent := FALSE, Sign := TRUE, MinLen := SINT#5, DecPlace := SINT#2);
(* Rung 7: Create STRING from Floating point coordinates *)
Attach := AddDelimiter(In := AttachPoint_STR, Delimiter := _COMMA);
(* Rung 8 *)
Vision_Result_OK := BYTE_TO_DINT(In := Vision_IN[60]);

(* Section ProgLoadRoboDK: ladder, written here as Structured Text *)

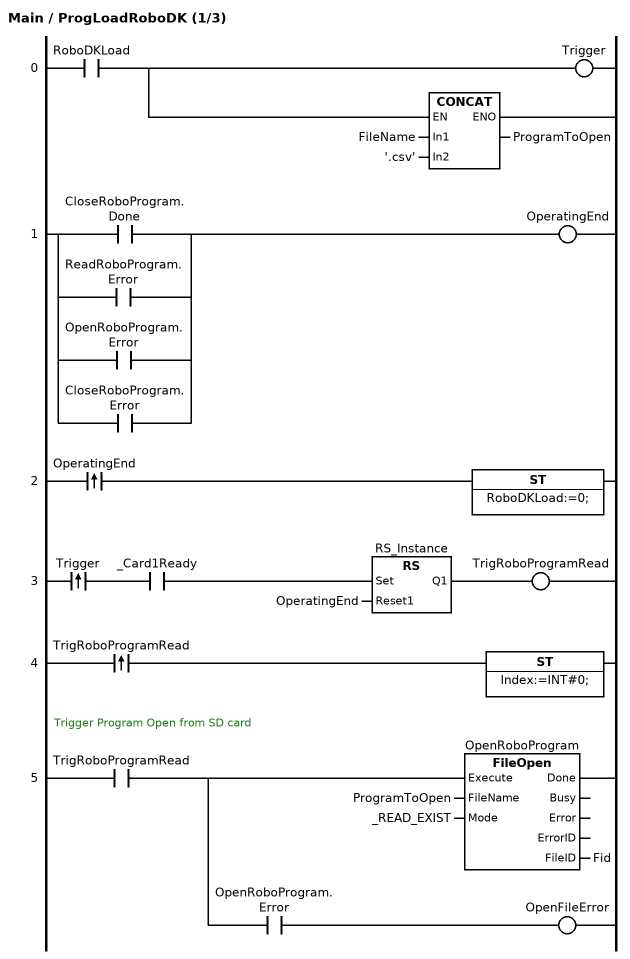
(* Rung 0 *)
Trigger := RoboDKLoad;
IF RoboDKLoad THEN ProgramToOpen := CONCAT(In1 := FileName, In2 := '.csv'); END_IF;
(* Rung 1 *)
OperatingEnd := CloseRoboProgram.Done OR ReadRoboProgram.Error OR OpenRoboProgram.Error OR CloseRoboProgram.Error;
(* Rung 2 *)
_e19(CLK := OperatingEnd);
IF _e19.Q THEN
    RoboDKLoad:=0;
END_IF;
(* Rung 3 *)
_e20(CLK := Trigger);
RS_Instance(Set := _e20.Q AND _Card1Ready, Reset1 := OperatingEnd);
TrigRoboProgramRead := RS_Instance.Q1;
(* Rung 4 *)
_e21(CLK := TrigRoboProgramRead);
IF _e21.Q THEN
    Index:=INT#0;
END_IF;
(* Rung 5: Trigger Program Open from SD card *)
OpenRoboProgram(Execute := TrigRoboProgramRead, FileName := ProgramToOpen, Mode := _READ_EXIST, FileID => Fid);
OpenFileError := TrigRoboProgramRead AND OpenRoboProgram.Error;

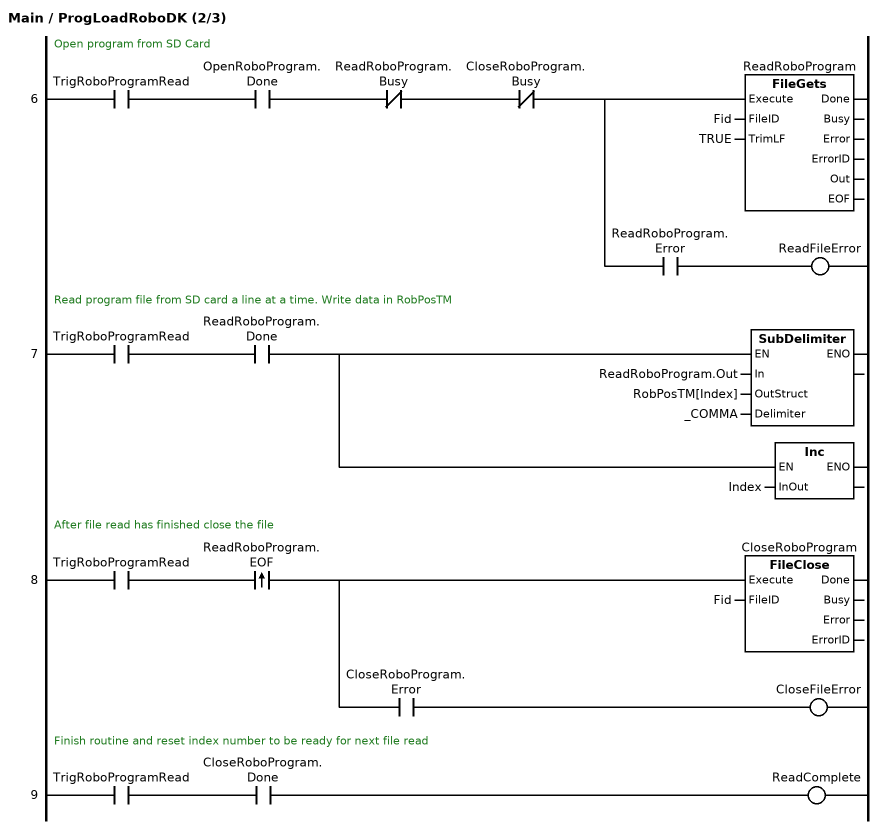
(* Rung 6: Open program from SD Card *)
_p22 := TrigRoboProgramRead AND OpenRoboProgram.Done AND NOT ReadRoboProgram.Busy AND NOT CloseRoboProgram.Busy;
ReadRoboProgram(Execute := _p22, FileID := Fid, TrimLF := TRUE);
ReadFileError := _p22 AND ReadRoboProgram.Error;
(* Rung 7: Read program file from SD card a line at a time. Write data in RobPosTM *)
_p23 := TrigRoboProgramRead AND ReadRoboProgram.Done;
IF _p23 THEN
    SubDelimiter(In := ReadRoboProgram.Out, OutStruct := RobPosTM[Index], Delimiter := _COMMA);
    Inc(InOut := Index);
END_IF;
(* Rung 8: After file read has finished close the file *)
_e24(CLK := ReadRoboProgram.EOF);
CloseRoboProgram(Execute := TrigRoboProgramRead AND _e24.Q, FileID := Fid);
CloseFileError := TrigRoboProgramRead AND _e24.Q AND CloseRoboProgram.Error;
(* Rung 9: Finish routine and reset index number to be ready for next file read *)
ReadComplete := TrigRoboProgramRead AND CloseRoboProgram.Done;

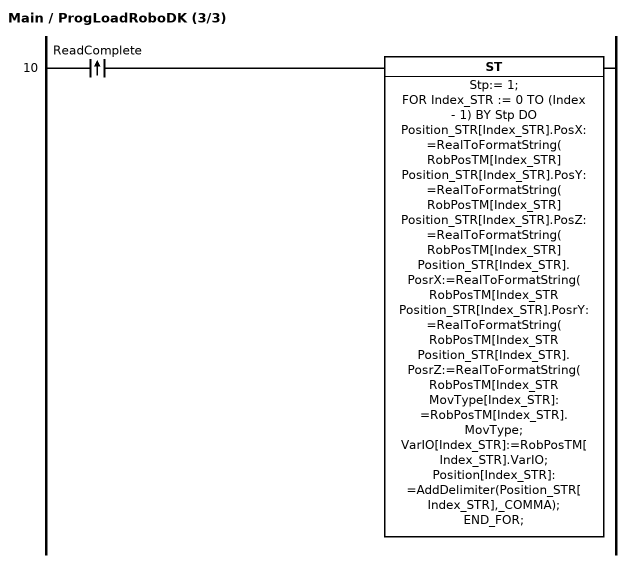
(* Rung 10 *)
_e25(CLK := ReadComplete);
IF _e25.Q THEN
    Stp:= 1;
    FOR Index_STR := 0 TO (Index - 1) BY Stp DO
    	Position_STR[Index_STR].PosX:=RealToFormatString(RobPosTM[Index_STR].RobPosX,FALSE,TRUE,SINT#5,SINT#2);
    	Position_STR[Index_STR].PosY:=RealToFormatString(RobPosTM[Index_STR].RobPosY,FALSE,TRUE,SINT#5,SINT#2);
    	Position_STR[Index_STR].PosZ:=RealToFormatString(RobPosTM[Index_STR].RobPosZ,FALSE,TRUE,SINT#5,SINT#2);
    	Position_STR[Index_STR].PosrX:=RealToFormatString(RobPosTM[Index_STR].RobPosrX,FALSE,TRUE,SINT#5,SINT#2);
    	Position_STR[Index_STR].PosrY:=RealToFormatString(RobPosTM[Index_STR].RobPosrY,FALSE,TRUE,SINT#5,SINT#2);
    	Position_STR[Index_STR].PosrZ:=RealToFormatString(RobPosTM[Index_STR].RobPosrZ,FALSE,TRUE,SINT#5,SINT#2);
    	MovType[Index_STR]:=RobPosTM[Index_STR].MovType;
    	VarIO[Index_STR]:=RobPosTM[Index_STR].VarIO;
    	Position[Index_STR]:=AddDelimiter(Position_STR[Index_STR],_COMMA);
    	
    END_FOR;
END_IF;

(* Section TapingMachine: ladder, written here as Structured Text *)

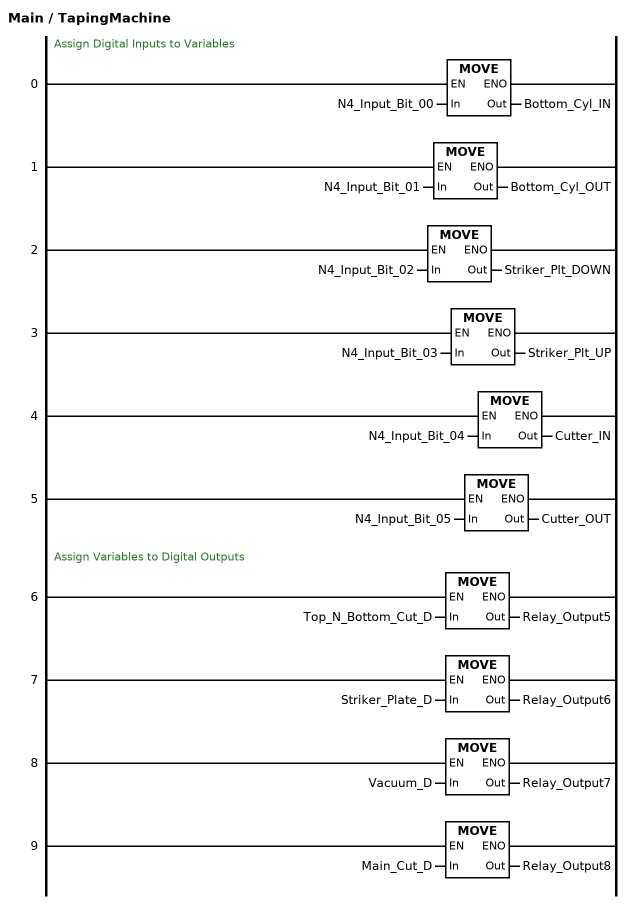
(* Rung 0: Assign Digital Inputs to Variables *)
Bottom_Cyl_IN := N4_Input_Bit_00;
(* Rung 1 *)
Bottom_Cyl_OUT := N4_Input_Bit_01;
(* Rung 2 *)
Striker_Plt_DOWN := N4_Input_Bit_02;
(* Rung 3 *)
Striker_Plt_UP := N4_Input_Bit_03;
(* Rung 4 *)
Cutter_IN := N4_Input_Bit_04;
(* Rung 5 *)
Cutter_OUT := N4_Input_Bit_05;
(* Rung 6: Assign Variables to Digital Outputs *)
Relay_Output5 := Top_N_Bottom_Cut_D;
(* Rung 7 *)
Relay_Output6 := Striker_Plate_D;
(* Rung 8 *)
Relay_Output7 := Vacuum_D;
(* Rung 9 *)
Relay_Output8 := Main_Cut_D;

(* Section ExtraIOMapping: ladder, written here as Structured Text *)

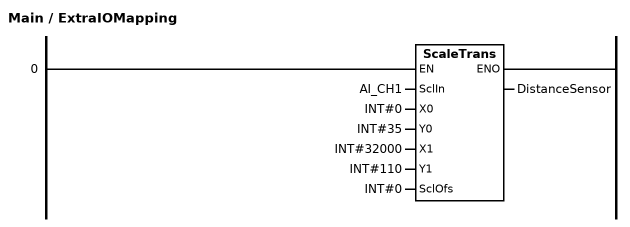
(* Rung 0 *)
DistanceSensor := ScaleTrans(SclIn := AI_CH1, X0 := INT#0, Y0 := INT#35, X1 := INT#32000, Y1 := INT#110, SclOfs := INT#0);

(* Section ERPConn: ladder, written here as Structured Text *)

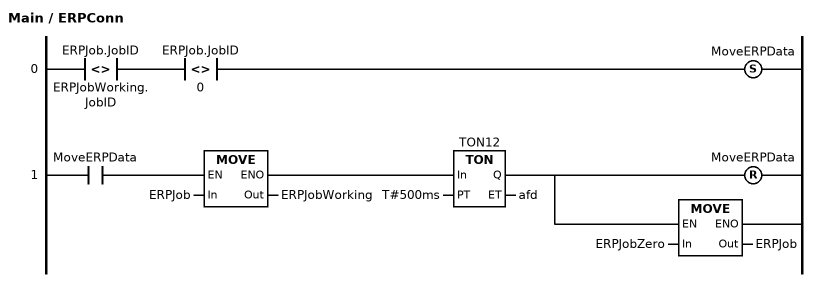
(* Rung 0 *)
IF (ERPJob.JobID <> ERPJobWorking.JobID) AND (ERPJob.JobID <> 0) THEN MoveERPData := TRUE; END_IF;
(* Rung 1 *)
IF MoveERPData THEN ERPJobWorking := ERPJob; END_IF;
TON12(In := MoveERPData, PT := T#500ms, ET => afd);
IF TON12.Q THEN
    MoveERPData := FALSE;
    ERPJob := ERPJobZero;
END_IF;
END_PROGRAM

PROGRAM TM_Movements_Connection
VAR
    ListenNode_Connect_Instance : ListenNode_Connect;
    ListenNode_Connect_Enable : BOOL;
    ListenNode_Connect_IPaddress : STRING[16];
    ListenNode_Connect_Port : UINT;
    ListenNode_Connect_Connect : BOOL;
    ListenNode_Connect_Error : BOOL;
    ListenNode_Connect_ErrorID : WORD;
    ListenNode_Connect_EtnConnError : BOOL;
    ListenNode_Connect_Socket_Status : _eCONNECTION_STATE;
END_VAR
VAR_EXTERNAL
    ListenNode_Connect_Connected : BOOL;
    ListenNode_Connect_TCP_Socket : _sSOCKET;
    StartProgram : BOOL;
END_VAR
ListenNode_Connect_Enable:=TRUE;
ListenNode_Connect_IPaddress:='10.1.20.60';
ListenNode_Connect_Port:=5890;

ListenNode_Connect_Connect:=StartProgram;

ListenNode_Connect_Instance(
	Enable:=ListenNode_Connect_Enable,
	IPaddress:=ListenNode_Connect_IPaddress,
	Port:=ListenNode_Connect_Port,
	Connect:=ListenNode_Connect_Connect,
	Connected=>ListenNode_Connect_Connected,
	Error=>ListenNode_Connect_Error,
	ErrorID=>ListenNode_Connect_ErrorID,
	EtnConnError=>ListenNode_Connect_EtnConnError,
	TCP_Socket=>ListenNode_Connect_TCP_Socket,
	Socket_Status=>ListenNode_Connect_Socket_Status
);
END_PROGRAM

PROGRAM TM_Movements
VAR
    TM_ChangeLoad_Instance : TM_ChangeLoad;
    TM_ChangeTCP_Instance : TM_ChangeTCP;
    TM_MovCmd_Instance : TM_MovCmd;
    TM_MovCmd_Done : BOOL;
    TM_MovCmd_Busy : BOOL;
    TM_MovCmd_Error : BOOL;
    TM_MovCmd_ErrorID : WORD;
    TM_MovCmd_Execute : BOOL;
    TM_MovCmd_Movement : STRING[256];
    TM_MovCmd_DataFormat : STRING[256];
    DD_ListenNode_Connect_Connected : F_TRIG;
    TM_MovCmd_Point : STRING[256];
    TM_MovCmd_Speed : INT;
    TM_MovCmd_AccelTime : INT;
    TM_MovCmd_Blending : INT;
    TM_MovCmd_PrecisePos : BOOL;
    TM_MovCmd_RobotPose : STRING[256];
    TM_MovCmd_ActivateExit : BOOL;
    TM_MovCmd_CommandID : INT;
    Enable : BOOL;
    DU_Enable : R_TRIG;
    TM_ChangeBase_Busy : BOOL;
    TM_ChangeBase_Done : BOOL;
    TM_ChangeBase_Error : BOOL;
    TM_ChangeBase_ErrorID : WORD;
    TM_ChangeBase_Execute : BOOL;
    TM_ChangeBase_Base : STRING[256];
    TM_ChangeBase_ActivateExit : BOOL;
    TM_ChangeBase_CommandID : INT;
    TM_ChangeLoad_Execute : BOOL;
    TM_ChangeLoad_Busy : BOOL;
    TM_ChangeLoad_Done : BOOL;
    TM_ChangeLoad_Error : BOOL;
    TM_ChangeLoad_ErrorID : WORD;
    TM_ChangeLoad_Payload : STRING[256];
    TM_ChangeLoad_ActivateExit : BOOL;
    TM_ChangeLoad_CommandID : INT;
    TM_ChangeTCP_Busy : BOOL;
    TM_ChangeTCP_Done : BOOL;
    TM_ChangeTCP_Error : BOOL;
    TM_ChangeTCP_ErrorID : WORD;
    TM_ChangeTCP_Execute : BOOL;
    TM_ChangeTCP_TCP : STRING[256];
    TM_ChangeTCP_Weight : STRING[256];
    TM_ChangeTCP_MomInertia : STRING[256];
    TM_ChangeTCP_RefFrame : STRING[256];
    TM_ChangeTCP_ActivateExit : BOOL;
    TM_ChangeTCP_CommandID : INT;
    TM_CircleCmd_Done : BOOL;
    TM_CircleCmd_Busy : BOOL;
    TM_CircleCmd_Error : BOOL;
    TM_CircleCmd_ErrorID : WORD;
    TM_CircleCmd_Execute : BOOL;
    TM_CircleCmd_DataFormat : STRING[256];
    TM_CircleCmd_ArcPoint : STRING[256];
    TM_CircleCmd_EndArcPoint : STRING[256];
    TM_CircleCmd_Speed : INT;
    TM_CircleCmd_AccelTime : INT;
    TM_CircleCmd_Blending : INT;
    TM_CircleCmd_ArcAngle : INT;
    TM_CircleCmd_PrecisePos : BOOL;
    TM_CircleCmd_Command : STRING[256];
    TM_CircleCmd_ActivateExit : BOOL;
    TM_CircleCmd_CommandID : INT;
    PickPoint : STRING[256];
    PalletFirstPoint : STRING[256];
    StartPoint : STRING[256];
    PalletSecondPoint : STRING[256];
    PalletThirdPoint : STRING[256];
    PalletFourthPoint : STRING[256];
    MovementIndicatorStage : INT;
    DownRelative : STRING[256];
    HighRelative : STRING[256];
    TM_ChangeBase_Command : STRING[256];
    TM_ChangeLoad_Command : STRING[256];
    TM_ChangeTCP_Command : STRING[256];
    DD_CableConnected : F_TRIG;
    TM_MovCmd_ListenNode : STRING[256];
    Stage : INT;
    TM_MovCmd_TimeOutET : TIME;
    TM_MovCmd_Enable : BOOL;
    TM_ChangeTCP_Enable : BOOL;
    TM_ChangeTCP_ListenNode : STRING[256];
    TM_ChangeTCP_TimeOutET : TIME;
    TM_ChangeLoad_Enable : BOOL;
    TM_ChangeLoad_ListenNode : STRING[256];
    TM_ChangeLoad_TimeOutET : TIME;
    TM_CircleCmd_Instance : TM_CircleCmd;
    TM_ChangeBase_Instance : TM_ChangeBase;
    TM_ChangeBase_Enable : BOOL;
    TM_CircleCmd_Enable : BOOL;
    TM_CircleCmd_ListenNode : STRING[256];
    TM_CircleCmd_TimeOutET : TIME;
    TM_ChangeBase_ListenNode : STRING[256];
    TM_ChangeBase_TimeOutET : TIME;
    Home : STRING[256];
    Midpoint : STRING[256];
    Approach : STRING[256];
    Position3 : STRING[256];
    Position2 : STRING[256];
    Position4 : STRING[256];
    Position5 : STRING[256];
    Position6 : STRING[256];
    Position7 : STRING[256];
    Position8 : STRING[256];
    Position9 : STRING[256];
    Position10 : STRING[256];
    Position11 : STRING[256];
    Rz_Attach_Original : REAL;
    Position12 : STRING[256];
    Midpoint1 : STRING[256];
    Approach1 : STRING[256];
    StepMove : INT;
END_VAR
VAR_EXTERNAL
    StartProgram : BOOL;
    CableConnected : BOOL;
    ListenNode_Connect_Connected : BOOL;
    ListenNode_Connect_TCP_Socket : _sSOCKET;
    Run_Stiching : BOOL;
    Stitching_Speed : REAL;
    Speed : REAL;
    TM_ReadPosition_X : REAL;
    TM_ReadPosition_Y : REAL;
    TM_ReadPosition_Z : REAL;
    TM_MovCmd_Command : STRING[256];
    RobPos_X : DINT;
    RobotIO : TMmodbus\sRobotIO;
    Stitching_InManual : BOOL;
    Part_Orientation_DINT : DINT;
    Vision_OUT : ARRAY[0..495] OF BYTE;
    RZ_Attach_String : STRING[256];
    Attach : STRING[256];
    Position1 : STRING[256];
    Position : ARRAY[0..100] OF STRING[100];
    MovType : ARRAY[0..100] OF STRING[100];
    RoboDKLoad : BOOL;
    FileName : STRING[100];
    ProgramToLoad : STRING[100];
    Index_STR : DINT;
    Run_Stiching_Man : BOOL;
    Stitcher_AutoSpeed : BOOL;
    Proj_Rob_Speed : INT;
    VarIO : ARRAY[0..100] OF STRING[100];
    Rob_Speed : DINT;
    Relay_Output9 : BOOL;
END_VAR
DU_Enable(Clk:=Enable);
DD_ListenNode_Connect_Connected(Clk:=ListenNode_Connect_Connected);
DD_CableConnected(Clk:=CableConnected);

Enable:=StartProgram;


IF DU_Enable.Q THEN
	
	Stage:=0;
	MovementIndicatorStage:=0;
	Proj_Rob_Speed:= 200;
	
END_IF;

IF DD_ListenNode_Connect_Connected.Q OR DD_CableConnected.Q THEN //connection closed or cable disconnected.
	
	Stage:= 9999; //MovementIndicatorStage;
	
END_IF;

IF Enable AND ListenNode_Connect_Connected AND CableConnected  THEN	//the PLC program is enabled and there is connection with listen node and the cable is connected
	 
	CASE Stage OF
				
		//-----------------------------------------------------------TCP Selection--------------------------------------------------
		0:
			TM_ChangeTCP_Enable:=FALSE;
			IF (NOT TM_ChangeTCP_Done) AND (NOT TM_ChangeTCP_Error) AND (NOT TM_ChangeTCP_Busy) THEN
				//FileName:= 'Prog1';
				//RoboDKLoad:=1;
				Stage:=1; 
			END_IF;
		1:	
			
			TM_ChangeTCP_Enable:=TRUE;	
			TM_ChangeTCP_ActivateExit:=TRUE;
			TM_ChangeTCP_CommandID:=1;
			TM_ChangeTCP_Execute:=FALSE;
			TM_ChangeTCP_ListenNode:='Listen1';
			TM_ChangeTCP_TCP:='Gripper';
			TM_MovCmd_Command:='var_switch=10'; //10 = pass; 20 = start stitching; 30 = stop stithing; 40 = gripper on; 50 = gripper off
			TM_ChangeTCP_Weight:='';
			TM_ChangeTCP_MomInertia:='';
			TM_ChangeTCP_RefFrame:='';
			TM_ChangeLoad_Payload:='';
			
			IF (NOT TM_ChangeTCP_Done) AND (NOT TM_ChangeTCP_Error) THEN
				
				Stage:=2;
				
			END_IF;
		2:
			TM_ChangeTCP_Execute:=TRUE;
			IF TM_ChangeTCP_Done THEN
				Stage:=10;
			ELSIF TM_ChangeTCP_Error THEN
				Stage:=9999;
			END_IF;
		//-----------------------------------------------------------Program Stages--------------------------------------------------------------
		10:
			TM_MovCmd_Enable:=FALSE;
			MovementIndicatorStage:=Stage;
			IF (NOT TM_MovCmd_Done) AND (NOT TM_MovCmd_Error) AND (NOT TM_MovCmd_Busy) THEN
				Stage:=11;
			END_IF;
		11:	
			StepMove:=1;
			TM_MovCmd_Enable:=TRUE;
			TM_MovCmd_Movement:= 'PTP';
			TM_MovCmd_Movement:= MovType[1];  //'PTP';
			IF MovType[1] = 'PTP'  THEN
			TM_MovCmd_DataFormat:='CPP';
			ELSE TM_MovCmd_DataFormat:='CPR';
			END_IF;
			TM_MovCmd_Point:=Position[1];
			TM_MovCmd_Speed:=Proj_Rob_Speed;
			TM_MovCmd_AccelTime:=200;
			TM_MovCmd_Blending:=0;
			TM_MovCmd_PrecisePos:=1;
			TM_MovCmd_RobotPose:='';
			IF VarIO[1] = '' THEN
			TM_MovCmd_Command:='var_switch=10'; //10 = pass; 20 = start stitching; 30 = stop stithing; 40 = gripper on; 50 = gripper off
			ELSE TM_MovCmd_Command:=VarIO[1];
			END_IF;
			TM_MovCmd_ActivateExit:=TRUE;
			TM_MovCmd_CommandID:=1;
			TM_MovCmd_Execute:=FALSE;
			TM_MovCmd_ListenNode:='Listen1';
			IF (NOT TM_MovCmd_Done) AND (NOT TM_MovCmd_Error) THEN
				Stage:=12;
			END_IF;
		12:
			TM_MovCmd_Execute:=TRUE;
			IF TM_MovCmd_Done AND Index_STR > 1 THEN
				
				Stage:=20;
			ELSIF TM_MovCmd_Error THEN
				Stage:=9999;
			END_IF;
		///////////////////////////////////////////////////////////////////////////////////////////////
		20:
			TM_MovCmd_Enable:=FALSE;
			MovementIndicatorStage:=Stage;
			IF (NOT TM_MovCmd_Done) AND (NOT TM_MovCmd_Error) AND (NOT TM_MovCmd_Busy) THEN
				Stage:=21;
			END_IF;
		21:			
			StepMove:=2;
			TM_MovCmd_Enable:=TRUE;
			TM_MovCmd_Movement:=MovType[2];
			IF MovType[2] = 'PTP'  THEN
			TM_MovCmd_DataFormat:='CPP';
			ELSE TM_MovCmd_DataFormat:='CPR';
			END_IF;
			TM_MovCmd_Point:=Position[2];
			TM_MovCmd_Speed:=Proj_Rob_Speed;
			TM_MovCmd_AccelTime:=200;
			TM_MovCmd_Blending:=0;
			TM_MovCmd_PrecisePos:=0;
			TM_MovCmd_RobotPose:='';
			IF VarIO[2] = '' THEN
			TM_MovCmd_Command:='var_switch=10'; //10 = pass; 20 = start stitching; 30 = stop stithing; 40 = gripper on; 50 = gripper off
			ELSE TM_MovCmd_Command:=VarIO[2];
			END_IF;
			TM_MovCmd_ActivateExit:=TRUE;
			TM_MovCmd_CommandID:=1;
			TM_MovCmd_Execute:=FALSE;
			TM_MovCmd_ListenNode:='Listen1';
			IF (NOT TM_MovCmd_Done) AND (NOT TM_MovCmd_Error) THEN
				Stage:=22;
			END_IF;			
		22:
			TM_MovCmd_Execute:=TRUE;
			IF TM_MovCmd_Done AND Index_STR > 2 THEN
				//////////////////////////////
				Stage:=30;
			ELSIF TM_MovCmd_Error THEN
				Stage:=9999;
			END_IF;
		///////////////////////////////////////////////////////////////////////////////////////////////
		30:
			TM_MovCmd_Enable:=FALSE;
			IF (NOT TM_MovCmd_Done) AND (NOT TM_MovCmd_Error) AND (NOT TM_MovCmd_Busy) THEN
				Stage:=31;
			END_IF;
		31:			
			StepMove:=3;
			TM_MovCmd_Enable:=TRUE;
			TM_MovCmd_Movement:=MovType[3];
			IF MovType[3] = 'PTP'  THEN
			TM_MovCmd_DataFormat:='CPP';
			ELSE TM_MovCmd_DataFormat:='CPR';
			END_IF;
			TM_MovCmd_Point:=Position[3];
			TM_MovCmd_Speed:=Proj_Rob_Speed;
			TM_MovCmd_AccelTime:=200;
			TM_MovCmd_Blending:=0;
			TM_MovCmd_PrecisePos:=1;
			TM_MovCmd_RobotPose:='';
			IF VarIO[3] = '' THEN
			TM_MovCmd_Command:='var_switch=20'; //10 = pass; 20 = start stitching; 30 = stop stithing; 40 = gripper on; 50 = gripper off
			ELSE TM_MovCmd_Command:=VarIO[3];
			END_IF;
			TM_MovCmd_ActivateExit:=TRUE;
			TM_MovCmd_CommandID:=1;
			TM_MovCmd_Execute:=FALSE;
			TM_MovCmd_ListenNode:='Listen1';
			IF (NOT TM_MovCmd_Done) AND (NOT TM_MovCmd_Error) THEN
				Stage:=32;
			END_IF;
		
		32:
			TM_MovCmd_Execute:=TRUE;
			IF TM_MovCmd_Done AND Index_STR > 3 THEN
				Stage:=40;
			ELSIF TM_MovCmd_Error THEN
				Stage:=9999;
			END_IF;
		///////////////////////////////////////////////////////////////////////////////////////////////	
		40:
			TM_MovCmd_Enable:=FALSE;
			IF (NOT TM_MovCmd_Done) AND (NOT TM_MovCmd_Error) AND (NOT TM_MovCmd_Busy) THEN
				Stage:=41;
			END_IF;	
		41:
			StepMove:=4;
			TM_MovCmd_Enable:=TRUE;
			TM_MovCmd_Movement:=MovType[4];
			IF MovType[4] = 'PTP'  THEN
			TM_MovCmd_DataFormat:='CPP';
			ELSE TM_MovCmd_DataFormat:='CPR';
			END_IF;
			TM_MovCmd_Point:=Position[4];
			TM_MovCmd_Speed:=Proj_Rob_Speed;
			TM_MovCmd_AccelTime:=200;
			TM_MovCmd_Blending:=0;
			TM_MovCmd_PrecisePos:=1;
			TM_MovCmd_RobotPose:='';
			IF VarIO[4] = '' THEN
			TM_MovCmd_Command:='var_switch=30'; //10 = pass; 20 = start stitching; 30 = stop stithing; 40 = gripper on; 50 = gripper off
			ELSE TM_MovCmd_Command:=VarIO[4];
			END_IF;
			TM_MovCmd_ActivateExit:=TRUE;
			TM_MovCmd_CommandID:=1;
			TM_MovCmd_Execute:=FALSE;
			TM_MovCmd_ListenNode:='Listen1';
			IF (NOT TM_MovCmd_Done) AND (NOT TM_MovCmd_Error) THEN
				Stage:=42;
			END_IF;
		42:
			TM_MovCmd_Execute:=TRUE;
			IF TM_MovCmd_Done AND Index_STR > 4 THEN
				Stage:=50;
			ELSIF TM_MovCmd_Error THEN
				Stage:=9999;
			END_IF;
		///////////////////////////////////////////////////////////////////////////////////////////////
		50:
			TM_MovCmd_Enable:=FALSE;
			MovementIndicatorStage:=Stage;
			IF (NOT TM_MovCmd_Done) AND (NOT TM_MovCmd_Error) AND (NOT TM_MovCmd_Busy) THEN
				Stage:=51;
			END_IF;	
		
		51:
			StepMove:=5;
			TM_MovCmd_Enable:=TRUE;
			TM_MovCmd_Movement:=MovType[5];
			IF MovType[5] = 'PTP'  THEN
			TM_MovCmd_DataFormat:='CPP';
			ELSE TM_MovCmd_DataFormat:='CPR';
			END_IF;
			TM_MovCmd_Point:=Position[5];
			TM_MovCmd_Speed:=Proj_Rob_Speed;
			TM_MovCmd_AccelTime:=200;
			TM_MovCmd_Blending:=0;
			TM_MovCmd_PrecisePos:=1;
			TM_MovCmd_RobotPose:='';
			IF VarIO[5] = '' THEN
			TM_MovCmd_Command:='var_switch=10'; //10 = pass; 20 = start stitching; 30 = stop stithing; 40 = gripper on; 50 = gripper off
			ELSE TM_MovCmd_Command:=VarIO[5];
			END_IF;
			TM_MovCmd_ActivateExit:=TRUE;
			TM_MovCmd_CommandID:=1;
			TM_MovCmd_Execute:=FALSE;
			TM_MovCmd_ListenNode:='Listen1';
			IF (NOT TM_MovCmd_Done) AND (NOT TM_MovCmd_Error) THEN
				Stage:=52;
			END_IF;
		52:
			TM_MovCmd_Execute:=TRUE;
			IF TM_MovCmd_Done AND Index_STR > 5 THEN
				Stage:=60;
			ELSIF TM_MovCmd_Error THEN
				Stage:=9999;
			END_IF;
		///////////////////////////////////////////////////////////////////////////////////////////////	
		60:
			TM_MovCmd_Enable:=FALSE;
			MovementIndicatorStage:=Stage;
			IF (NOT TM_MovCmd_Done) AND (NOT TM_MovCmd_Error) AND (NOT TM_MovCmd_Busy) THEN
				Stage:=61;
			END_IF;	
		
		61:
			StepMove:=6;
			TM_MovCmd_Enable:=TRUE;
			TM_MovCmd_Movement:=MovType[6];
			IF MovType[6] = 'PTP'  THEN
			TM_MovCmd_DataFormat:='CPP';
			ELSE TM_MovCmd_DataFormat:='CPR';
			END_IF;
			TM_MovCmd_Point:=Position[6];
			TM_MovCmd_Speed:=Proj_Rob_Speed;
			TM_MovCmd_AccelTime:=200;
			TM_MovCmd_Blending:=0;
			TM_MovCmd_PrecisePos:=0;
			TM_MovCmd_RobotPose:='';
			IF VarIO[6] = '' THEN
			TM_MovCmd_Command:='var_switch=10'; //10 = pass; 20 = start stitching; 30 = stop stithing; 40 = gripper on; 50 = gripper off
			ELSE TM_MovCmd_Command:=VarIO[6];
			END_IF;
			TM_MovCmd_ActivateExit:=TRUE;
			TM_MovCmd_CommandID:=1;
			TM_MovCmd_Execute:=FALSE;
			TM_MovCmd_ListenNode:='Listen1';
			IF (NOT TM_MovCmd_Done) AND (NOT TM_MovCmd_Error) THEN
				Stage:=62;
			END_IF;
		62:
			TM_MovCmd_Execute:=TRUE;
			IF TM_MovCmd_Done AND Index_STR > 6 THEN
				Stage:=70;
			ELSIF TM_MovCmd_Error THEN
				Stage:=9999;
			END_IF;
		///////////////////////////////////////////////////////////////////////////////////////////////
		70:
			TM_MovCmd_Enable:=FALSE;
			MovementIndicatorStage:=Stage;
			IF (NOT TM_MovCmd_Done) AND (NOT TM_MovCmd_Error) AND (NOT TM_MovCmd_Busy) THEN
				Stage:=71;
			END_IF;	
		
		71:
			StepMove:=7;
			TM_MovCmd_Enable:=TRUE;
			TM_MovCmd_Movement:=MovType[7];
			IF MovType[7] = 'PTP'  THEN
			TM_MovCmd_DataFormat:='CPP';
			ELSE TM_MovCmd_DataFormat:='CPR';
			END_IF;
			TM_MovCmd_Point:=Position[7];
			TM_MovCmd_Speed:=Proj_Rob_Speed;
			TM_MovCmd_AccelTime:=200;
			TM_MovCmd_Blending:=0;
			TM_MovCmd_PrecisePos:=0;
			TM_MovCmd_RobotPose:='';
			IF VarIO[7] = '' THEN
			TM_MovCmd_Command:='var_switch=20'; //10 = pass; 20 = start stitching; 30 = stop stithing; 40 = gripper on; 50 = gripper off
			ELSE TM_MovCmd_Command:=VarIO[7];
			END_IF;
			TM_MovCmd_ActivateExit:=TRUE;
			TM_MovCmd_CommandID:=1;
			TM_MovCmd_Execute:=FALSE;
			TM_MovCmd_ListenNode:='Listen1';
			IF (NOT TM_MovCmd_Done) AND (NOT TM_MovCmd_Error) THEN
				Stage:=72;
			END_IF;
		72:
			TM_MovCmd_Execute:=TRUE;
			IF TM_MovCmd_Done AND Index_STR > 7 THEN
				Stage:=80;
			ELSIF TM_MovCmd_Error THEN
				Stage:=9999;
			END_IF;
		///////////////////////////////////////////////////////////////////////////////////////////////
		80:
			TM_MovCmd_Enable:=FALSE;
			MovementIndicatorStage:=Stage;
			IF (NOT TM_MovCmd_Done) AND (NOT TM_MovCmd_Error) AND (NOT TM_MovCmd_Busy) THEN
				Stage:=81;
			END_IF;	
		
		81:
			StepMove:=8;
			TM_MovCmd_Enable:=TRUE;
			TM_MovCmd_Movement:=MovType[8];
			IF MovType[8] = 'PTP'  THEN
			TM_MovCmd_DataFormat:='CPP';
			ELSE TM_MovCmd_DataFormat:='CPR';
			END_IF;
			TM_MovCmd_Point:=Position[8];
			TM_MovCmd_Speed:=Proj_Rob_Speed;
			TM_MovCmd_AccelTime:=200;
			TM_MovCmd_Blending:=0;
			TM_MovCmd_PrecisePos:=1;
			TM_MovCmd_RobotPose:='';
			IF VarIO[8] = '' THEN
			TM_MovCmd_Command:='var_switch=30'; //10 = pass; 20 = start stitching; 30 = stop stithing; 40 = gripper on; 50 = gripper off
			ELSE TM_MovCmd_Command:=VarIO[8];
			END_IF;
			TM_MovCmd_ActivateExit:=TRUE;
			TM_MovCmd_CommandID:=1;
			TM_MovCmd_Execute:=FALSE;
			TM_MovCmd_ListenNode:='Listen1';
		
			IF (NOT TM_MovCmd_Done) AND (NOT TM_MovCmd_Error) THEN
				Stage:=82;
			END_IF;
		82:
			TM_MovCmd_Execute:=TRUE;
			IF TM_MovCmd_Done AND Index_STR > 8 THEN
				Stage:=90;
			ELSIF TM_MovCmd_Error THEN
				Stage:=9999;
			END_IF;	
			///////////////////////////////////////////////////////////////////////////////////////////////
		90:
			TM_MovCmd_Enable:=FALSE;
			MovementIndicatorStage:=Stage;
			IF (NOT TM_MovCmd_Done) AND (NOT TM_MovCmd_Error) AND (NOT TM_MovCmd_Busy) THEN
				Stage:=91;
			END_IF;	
		
		91:
			StepMove:=9;
			TM_MovCmd_Enable:=TRUE;
			TM_MovCmd_Movement:=MovType[9];
			IF MovType[9] = 'PTP'  THEN
			TM_MovCmd_DataFormat:='CPP';
			ELSE TM_MovCmd_DataFormat:='CPR';
			END_IF;
			TM_MovCmd_Point:=Position[9];
			TM_MovCmd_Speed:=Proj_Rob_Speed;
			TM_MovCmd_AccelTime:=200;
			TM_MovCmd_Blending:=0;
			TM_MovCmd_PrecisePos:=1;
			TM_MovCmd_RobotPose:='';
			IF VarIO[9] = '' THEN
			TM_MovCmd_Command:='var_switch=10'; //10 = pass; 20 = start stitching; 30 = stop stithing; 40 = gripper on; 50 = gripper off
			ELSE TM_MovCmd_Command:=VarIO[9];
			END_IF;
			TM_MovCmd_ActivateExit:=TRUE;
			TM_MovCmd_CommandID:=1;
			TM_MovCmd_Execute:=FALSE;
			TM_MovCmd_ListenNode:='Listen1';
		
			IF (NOT TM_MovCmd_Done) AND (NOT TM_MovCmd_Error) THEN
				Stage:=92;
			END_IF;
		92:
			TM_MovCmd_Execute:=TRUE;
			IF TM_MovCmd_Done AND Index_STR > 9 THEN
				Stage:=100;
			ELSIF TM_MovCmd_Error THEN
				Stage:=9999;
			END_IF;
			///////////////////////////////////////////////////////////////////////////////////////////////
			100:
			TM_MovCmd_Enable:=FALSE;
			MovementIndicatorStage:=Stage;
			IF (NOT TM_MovCmd_Done) AND (NOT TM_MovCmd_Error) AND (NOT TM_MovCmd_Busy) THEN
				Stage:=101;
			END_IF;	
		
		101:
			StepMove:=10;
			TM_MovCmd_Enable:=TRUE;
			TM_MovCmd_Movement:=MovType[10];
			IF MovType[10] = 'PTP'  THEN
			TM_MovCmd_DataFormat:='CPP';
			ELSE TM_MovCmd_DataFormat:='CPR';
			END_IF;
			TM_MovCmd_Point:=Position[10];
			TM_MovCmd_Speed:=Proj_Rob_Speed;
			TM_MovCmd_AccelTime:=200;
			TM_MovCmd_Blending:=0;
			TM_MovCmd_PrecisePos:=1;
			TM_MovCmd_RobotPose:='';
			IF VarIO[10] = '' THEN
			TM_MovCmd_Command:='var_switch=10'; //10 = pass; 20 = start stitching; 30 = stop stithing; 40 = gripper on; 50 = gripper off
			ELSE TM_MovCmd_Command:=VarIO[10];
			END_IF;
			TM_MovCmd_ActivateExit:=TRUE;
			TM_MovCmd_CommandID:=1;
			TM_MovCmd_Execute:=FALSE;
			TM_MovCmd_ListenNode:='Listen1';
		
			IF (NOT TM_MovCmd_Done) AND (NOT TM_MovCmd_Error) THEN
				Stage:=102;
			END_IF;
		
		102:
			TM_MovCmd_Execute:=TRUE;
			IF TM_MovCmd_Done AND Index_STR > 10 THEN
				Stage:=110;
			ELSIF TM_MovCmd_Error THEN
				Stage:=9999;
			END_IF;
			///////////////////////////////////////////////////////////////////////////////////////////////
			110:
			TM_MovCmd_Enable:=FALSE;
			MovementIndicatorStage:=Stage;
			IF (NOT TM_MovCmd_Done) AND (NOT TM_MovCmd_Error) AND (NOT TM_MovCmd_Busy) THEN
				Stage:=111;
			END_IF;	
		
		111:
			StepMove:=11;
			TM_MovCmd_Enable:=TRUE;
			TM_MovCmd_Movement:=MovType[11];
			IF MovType[11] = 'PTP'  THEN
			TM_MovCmd_DataFormat:='CPP';
			ELSE TM_MovCmd_DataFormat:='CPR';
			END_IF;
			TM_MovCmd_Point:=Position[11];
			TM_MovCmd_Speed:=Proj_Rob_Speed;
			TM_MovCmd_AccelTime:=200;
			TM_MovCmd_Blending:=0;
			TM_MovCmd_PrecisePos:=1;
			TM_MovCmd_RobotPose:='';
			IF VarIO[11] = '' THEN
			TM_MovCmd_Command:='var_switch=20'; //10 = pass; 20 = start stitching; 30 = stop stithing; 40 = gripper on; 50 = gripper off
			ELSE TM_MovCmd_Command:=VarIO[11];
			END_IF;
			TM_MovCmd_ActivateExit:=TRUE;
			TM_MovCmd_CommandID:=1;
			TM_MovCmd_Execute:=FALSE;
			TM_MovCmd_ListenNode:='Listen1';
		
			IF (NOT TM_MovCmd_Done) AND (NOT TM_MovCmd_Error) THEN
				Stage:=112;
			END_IF;
		112:
			TM_MovCmd_Execute:=TRUE;
			IF TM_MovCmd_Done AND Index_STR > 11 THEN
				Stage:=120;
			ELSIF TM_MovCmd_Error THEN
				Stage:=9999;
			END_IF;
		120:
			TM_MovCmd_Enable:=FALSE;
			MovementIndicatorStage:=Stage;
			IF (NOT TM_MovCmd_Done) AND (NOT TM_MovCmd_Error) AND (NOT TM_MovCmd_Busy) THEN
				Stage:=121;
			END_IF;	
		
		121:
			StepMove:=12;
			TM_MovCmd_Enable:=TRUE;
			TM_MovCmd_Movement:=MovType[12];
			IF MovType[12] = 'PTP'  THEN
			TM_MovCmd_DataFormat:='CPP';
			ELSE TM_MovCmd_DataFormat:='CPR';
			END_IF;
			TM_MovCmd_Point:=Position[12];
			TM_MovCmd_Speed:=Proj_Rob_Speed;
			TM_MovCmd_AccelTime:=200;
			TM_MovCmd_Blending:=0;
			TM_MovCmd_PrecisePos:=1;
			TM_MovCmd_RobotPose:='';
			IF VarIO[12] = '' THEN
			TM_MovCmd_Command:='var_switch=30'; //10 = pass; 20 = start stitching; 30 = stop stithing; 40 = gripper on; 50 = gripper off
			ELSE TM_MovCmd_Command:=VarIO[12];
			END_IF;
			TM_MovCmd_ActivateExit:=TRUE;
			TM_MovCmd_CommandID:=1;
			TM_MovCmd_Execute:=FALSE;
			TM_MovCmd_ListenNode:='Listen1';
		
			IF (NOT TM_MovCmd_Done) AND (NOT TM_MovCmd_Error) THEN
				Stage:=122;
			END_IF;
		122:
			TM_MovCmd_Execute:=TRUE;
			IF TM_MovCmd_Done AND Index_STR > 12 THEN
				Stage:=130;
			ELSIF TM_MovCmd_Error THEN
				Stage:=9999;
			END_IF;	
			///////////////////////////////////////////////////////////////////////////////////////////////
		130:
			TM_MovCmd_Enable:=FALSE;
			MovementIndicatorStage:=Stage;
			IF (NOT TM_MovCmd_Done) AND (NOT TM_MovCmd_Error) AND (NOT TM_MovCmd_Busy) THEN
				Stage:=131;
			END_IF;	
		
		131:
			StepMove:=13;
			TM_MovCmd_Enable:=TRUE;
			TM_MovCmd_Movement:=MovType[13];
			IF MovType[13] = 'PTP'  THEN
			TM_MovCmd_DataFormat:='CPP';
			ELSE TM_MovCmd_DataFormat:='CPR';
			END_IF;
			TM_MovCmd_Point:=Position[13];
			TM_MovCmd_Speed:=Proj_Rob_Speed;
			TM_MovCmd_AccelTime:=200;
			TM_MovCmd_Blending:=0;
			TM_MovCmd_PrecisePos:=1;
			TM_MovCmd_RobotPose:='';
			IF VarIO[13] = '' THEN
			TM_MovCmd_Command:='var_switch=10'; //10 = pass; 20 = start stitching; 30 = stop stithing; 40 = gripper on; 50 = gripper off
			ELSE TM_MovCmd_Command:=VarIO[13];
			END_IF;
			TM_MovCmd_ActivateExit:=TRUE;
			TM_MovCmd_CommandID:=1;
			TM_MovCmd_Execute:=FALSE;
			TM_MovCmd_ListenNode:='Listen1';
		
			IF (NOT TM_MovCmd_Done) AND (NOT TM_MovCmd_Error) THEN
				Stage:=132;
			END_IF;
		132:
			TM_MovCmd_Execute:=TRUE;
			IF TM_MovCmd_Done AND Index_STR > 13 THEN
				Stage:=140;
			ELSIF TM_MovCmd_Error THEN
				Stage:=9999;
			END_IF;
			
		140:
			TM_MovCmd_Enable:=FALSE;
			MovementIndicatorStage:=Stage;
			IF (NOT TM_MovCmd_Done) AND (NOT TM_MovCmd_Error) AND (NOT TM_MovCmd_Busy) THEN
				Stage:=141;
			END_IF;	
		
		141:
			StepMove:=14;
			TM_MovCmd_Enable:=TRUE;
			TM_MovCmd_Movement:=MovType[14];
			IF MovType[14] = 'PTP'  THEN
			TM_MovCmd_DataFormat:='CPP';
			ELSE TM_MovCmd_DataFormat:='CPR';
			END_IF;
			TM_MovCmd_Point:=Position[14];
			TM_MovCmd_Speed:=Proj_Rob_Speed;
			TM_MovCmd_AccelTime:=200;
			TM_MovCmd_Blending:=0;
			TM_MovCmd_PrecisePos:=1;
			TM_MovCmd_RobotPose:='';
			IF VarIO[14] = '' THEN
			TM_MovCmd_Command:='var_switch=10'; //10 = pass; 20 = start stitching; 30 = stop stithing; 40 = gripper on; 50 = gripper off
			ELSE TM_MovCmd_Command:=VarIO[14];
			END_IF;
			TM_MovCmd_ActivateExit:=TRUE;
			TM_MovCmd_CommandID:=1;
			TM_MovCmd_Execute:=FALSE;
			TM_MovCmd_ListenNode:='Listen1';
		
			IF (NOT TM_MovCmd_Done) AND (NOT TM_MovCmd_Error) THEN
				Stage:=142;
			END_IF;
		
		142:
			TM_MovCmd_Execute:=TRUE;
			IF TM_MovCmd_Done AND Index_STR > 14 THEN
				Stage:=150;
			ELSIF TM_MovCmd_Error THEN
				Stage:=9999;
			END_IF;
			///////////////////////////////////////////////////////////////////////////////////////////////
		150:
			TM_MovCmd_Enable:=FALSE;
			MovementIndicatorStage:=Stage;
			IF (NOT TM_MovCmd_Done) AND (NOT TM_MovCmd_Error) AND (NOT TM_MovCmd_Busy) THEN
				Stage:=151;
			END_IF;	
		
		151:
			StepMove:=15;
			TM_MovCmd_Enable:=TRUE;
			TM_MovCmd_Movement:=MovType[15];
			IF MovType[15] = 'PTP'  THEN
			TM_MovCmd_DataFormat:='CPP';
			ELSE TM_MovCmd_DataFormat:='CPR';
			END_IF;
			TM_MovCmd_Point:=Position[15];
			TM_MovCmd_Speed:=Proj_Rob_Speed;
			TM_MovCmd_AccelTime:=200;
			TM_MovCmd_Blending:=0;
			TM_MovCmd_PrecisePos:=1;
			TM_MovCmd_RobotPose:='';
			IF VarIO[15] = '' THEN
			TM_MovCmd_Command:='var_switch=20'; //10 = pass; 20 = start stitching; 30 = stop stithing; 40 = gripper on; 50 = gripper off
			ELSE TM_MovCmd_Command:=VarIO[15];
			END_IF;
			TM_MovCmd_ActivateExit:=TRUE;
			TM_MovCmd_CommandID:=1;
			TM_MovCmd_Execute:=FALSE;
			TM_MovCmd_ListenNode:='Listen1';
		
			IF (NOT TM_MovCmd_Done) AND (NOT TM_MovCmd_Error) THEN
				Stage:=152;
			END_IF;
		152:
			TM_MovCmd_Execute:=TRUE;
			IF TM_MovCmd_Done AND Index_STR > 15 THEN
				Stage:=160;
			ELSIF TM_MovCmd_Error THEN
				Stage:=9999;
			END_IF;
			
		160:
			TM_MovCmd_Enable:=FALSE;
			MovementIndicatorStage:=Stage;
			IF (NOT TM_MovCmd_Done) AND (NOT TM_MovCmd_Error) AND (NOT TM_MovCmd_Busy) THEN
				Stage:=161;
			END_IF;	
		
		161:
			StepMove:=16;
			TM_MovCmd_Enable:=TRUE;
			TM_MovCmd_Movement:=MovType[16];
			IF MovType[16] = 'PTP'  THEN
			TM_MovCmd_DataFormat:='CPP';
			ELSE TM_MovCmd_DataFormat:='CPR';
			END_IF;
			TM_MovCmd_Point:=Position[16];
			TM_MovCmd_Speed:=Proj_Rob_Speed;
			TM_MovCmd_AccelTime:=200;
			TM_MovCmd_Blending:=0;
			TM_MovCmd_PrecisePos:=1;
			TM_MovCmd_RobotPose:='';
			IF VarIO[16] = '' THEN
			TM_MovCmd_Command:='var_switch=30'; //10 = pass; 20 = start stitching; 30 = stop stithing; 40 = gripper on; 50 = gripper off
			ELSE TM_MovCmd_Command:=VarIO[16];
			END_IF;
			TM_MovCmd_ActivateExit:=TRUE;
			TM_MovCmd_CommandID:=1;
			TM_MovCmd_Execute:=FALSE;
			TM_MovCmd_ListenNode:='Listen1';
		
			IF (NOT TM_MovCmd_Done) AND (NOT TM_MovCmd_Error) THEN
				Stage:=162;
			END_IF;
		162:
			TM_MovCmd_Execute:=TRUE;
			IF TM_MovCmd_Done AND Index_STR > 16 THEN
				Stage:=170;
			ELSIF TM_MovCmd_Error THEN
				Stage:=9999;
			END_IF;
		170:
			TM_MovCmd_Enable:=FALSE;
			MovementIndicatorStage:=Stage;
			IF (NOT TM_MovCmd_Done) AND (NOT TM_MovCmd_Error) AND (NOT TM_MovCmd_Busy) THEN
				Stage:=171;
			END_IF;	
		
		171:
			StepMove:=17;
			TM_MovCmd_Enable:=TRUE;
			TM_MovCmd_Movement:=MovType[17];
			IF MovType[17] = 'PTP'  THEN
			TM_MovCmd_DataFormat:='CPP';
			ELSE TM_MovCmd_DataFormat:='CPR';
			END_IF;
			TM_MovCmd_Point:=Position[17];
			TM_MovCmd_Speed:=Proj_Rob_Speed;
			TM_MovCmd_AccelTime:=200;
			TM_MovCmd_Blending:=0;
			TM_MovCmd_PrecisePos:=1;
			TM_MovCmd_RobotPose:='';
			IF VarIO[17] = '' THEN
			TM_MovCmd_Command:='var_switch=10'; //10 = pass; 20 = start stitching; 30 = stop stithing; 40 = gripper on; 50 = gripper off
			ELSE TM_MovCmd_Command:=VarIO[17];
			END_IF;
			TM_MovCmd_ActivateExit:=TRUE;
			TM_MovCmd_CommandID:=1;
			TM_MovCmd_Execute:=FALSE;
			TM_MovCmd_ListenNode:='Listen1';
		
			IF (NOT TM_MovCmd_Done) AND (NOT TM_MovCmd_Error) THEN
				Stage:=172;
			END_IF;
		172:
			TM_MovCmd_Execute:=TRUE;
			IF TM_MovCmd_Done AND Index_STR > 17 THEN
				Stage:=180;
			ELSIF TM_MovCmd_Error THEN
				Stage:=9999;
			END_IF;		
		180:
			TM_MovCmd_Enable:=FALSE;
			MovementIndicatorStage:=Stage;
			IF (NOT TM_MovCmd_Done) AND (NOT TM_MovCmd_Error) AND (NOT TM_MovCmd_Busy) THEN
				Stage:=181;
			END_IF;	
		
		181:
			StepMove:=18;
			TM_MovCmd_Enable:=TRUE;
			TM_MovCmd_Movement:=MovType[18];
			IF MovType[18] = 'PTP'  THEN
			TM_MovCmd_DataFormat:='CPP';
			ELSE TM_MovCmd_DataFormat:='CPR';
			END_IF;
			TM_MovCmd_Point:=Position[18];
			TM_MovCmd_Speed:=Proj_Rob_Speed;
			TM_MovCmd_AccelTime:=200;
			TM_MovCmd_Blending:=0;
			TM_MovCmd_PrecisePos:=1;
			TM_MovCmd_RobotPose:='';
			IF VarIO[18] = '' THEN
			TM_MovCmd_Command:='var_switch=10'; //10 = pass; 20 = start stitching; 30 = stop stithing; 40 = gripper on; 50 = gripper off
			ELSE TM_MovCmd_Command:=VarIO[18];
			END_IF;
			TM_MovCmd_ActivateExit:=TRUE;
			TM_MovCmd_CommandID:=1;
			TM_MovCmd_Execute:=FALSE;
			TM_MovCmd_ListenNode:='Listen1';
		
			IF (NOT TM_MovCmd_Done) AND (NOT TM_MovCmd_Error) THEN
				Stage:=182;
			END_IF;
		182:
			TM_MovCmd_Execute:=TRUE;
			IF TM_MovCmd_Done AND Index_STR > 18 THEN
				Stage:=190;
			ELSIF TM_MovCmd_Error THEN
				Stage:=9999;
			END_IF;	
		190:
			TM_MovCmd_Enable:=FALSE;
			MovementIndicatorStage:=Stage;
			IF (NOT TM_MovCmd_Done) AND (NOT TM_MovCmd_Error) AND (NOT TM_MovCmd_Busy) THEN
				Stage:=191;
			END_IF;	
		
		191:
			StepMove:=19;
			TM_MovCmd_Enable:=TRUE;
			TM_MovCmd_Movement:=MovType[19];
			IF MovType[19] = 'PTP'  THEN
			TM_MovCmd_DataFormat:='CPP';
			ELSE TM_MovCmd_DataFormat:='CPR';
			END_IF;
			TM_MovCmd_Point:=Position[19];
			TM_MovCmd_Speed:=Proj_Rob_Speed;
			TM_MovCmd_AccelTime:=200;
			TM_MovCmd_Blending:=0;
			TM_MovCmd_PrecisePos:=1;
			TM_MovCmd_RobotPose:='';
			IF VarIO[19] = '' THEN
			TM_MovCmd_Command:='var_switch=10'; //10 = pass; 20 = start stitching; 30 = stop stithing; 40 = gripper on; 50 = gripper off
			ELSE TM_MovCmd_Command:=VarIO[19];
			END_IF;
			TM_MovCmd_ActivateExit:=TRUE;
			TM_MovCmd_CommandID:=1;
			TM_MovCmd_Execute:=FALSE;
			TM_MovCmd_ListenNode:='Listen1';
		
			IF (NOT TM_MovCmd_Done) AND (NOT TM_MovCmd_Error) THEN
				Stage:=192;
			END_IF;
		192:
			TM_MovCmd_Execute:=TRUE;
			IF TM_MovCmd_Done AND Index_STR > 19 THEN
				Stage:=200;
			ELSIF TM_MovCmd_Error THEN
				Stage:=9999;
			END_IF;		
		200:
			TM_MovCmd_Enable:=FALSE;
			MovementIndicatorStage:=Stage;
			IF (NOT TM_MovCmd_Done) AND (NOT TM_MovCmd_Error) AND (NOT TM_MovCmd_Busy) THEN
				Stage:=201;
			END_IF;	
		
		201:
			StepMove:=20;
			TM_MovCmd_Enable:=TRUE;
			TM_MovCmd_Movement:=MovType[20];
			IF MovType[20] = 'PTP'  THEN
			TM_MovCmd_DataFormat:='CPP';
			ELSE TM_MovCmd_DataFormat:='CPR';
			END_IF;
			TM_MovCmd_Point:=Position[20];
			TM_MovCmd_Speed:=Proj_Rob_Speed;
			TM_MovCmd_AccelTime:=200;
			TM_MovCmd_Blending:=0;
			TM_MovCmd_PrecisePos:=1;
			TM_MovCmd_RobotPose:='';
			IF VarIO[20] = '' THEN
			TM_MovCmd_Command:='var_switch=10'; //10 = pass; 20 = start stitching; 30 = stop stithing; 40 = gripper on; 50 = gripper off
			ELSE TM_MovCmd_Command:=VarIO[20];
			END_IF;
			TM_MovCmd_ActivateExit:=TRUE;
			TM_MovCmd_CommandID:=1;
			TM_MovCmd_Execute:=FALSE;
			TM_MovCmd_ListenNode:='Listen1';
		
			IF (NOT TM_MovCmd_Done) AND (NOT TM_MovCmd_Error) THEN
				Stage:=202;
			END_IF;
		202:
			TM_MovCmd_Execute:=TRUE;
			IF TM_MovCmd_Done AND Index_STR > 20 THEN
				Stage:=210;
			ELSIF TM_MovCmd_Error THEN
				Stage:=9999;
			END_IF;		
		210:
			TM_MovCmd_Enable:=FALSE;
			MovementIndicatorStage:=Stage;
			IF (NOT TM_MovCmd_Done) AND (NOT TM_MovCmd_Error) AND (NOT TM_MovCmd_Busy) THEN
				Stage:=211;
			END_IF;	
		
		211:
			StepMove:=21;
			TM_MovCmd_Enable:=TRUE;
			TM_MovCmd_Movement:=MovType[21];
			IF MovType[21] = 'PTP'  THEN
			TM_MovCmd_DataFormat:='CPP';
			ELSE TM_MovCmd_DataFormat:='CPR';
			END_IF;
			TM_MovCmd_Point:=Position[21];
			TM_MovCmd_Speed:=Proj_Rob_Speed;
			TM_MovCmd_AccelTime:=200;
			TM_MovCmd_Blending:=0;
			TM_MovCmd_PrecisePos:=1;
			TM_MovCmd_RobotPose:='';
			IF VarIO[21] = '' THEN
			TM_MovCmd_Command:='var_switch=10'; //10 = pass; 20 = start stitching; 30 = stop stithing; 40 = gripper on; 50 = gripper off
			ELSE TM_MovCmd_Command:=VarIO[21];
			END_IF;
			TM_MovCmd_ActivateExit:=TRUE;
			TM_MovCmd_CommandID:=1;
			TM_MovCmd_Execute:=FALSE;
			TM_MovCmd_ListenNode:='Listen1';
		
			IF (NOT TM_MovCmd_Done) AND (NOT TM_MovCmd_Error) THEN
				Stage:=212;
			END_IF;
		212:
			TM_MovCmd_Execute:=TRUE;
			IF TM_MovCmd_Done AND Index_STR > 21 THEN
				Stage:=220;
			ELSIF TM_MovCmd_Error THEN
				Stage:=9999;
			END_IF;		
		220:
			TM_MovCmd_Enable:=FALSE;
			MovementIndicatorStage:=Stage;
			IF (NOT TM_MovCmd_Done) AND (NOT TM_MovCmd_Error) AND (NOT TM_MovCmd_Busy) THEN
				Stage:=221;
			END_IF;	
		
		221:
			StepMove:=22;
			TM_MovCmd_Enable:=TRUE;
			TM_MovCmd_Movement:=MovType[22];
			IF MovType[22] = 'PTP'  THEN
			TM_MovCmd_DataFormat:='CPP';
			ELSE TM_MovCmd_DataFormat:='CPR';
			END_IF;
			TM_MovCmd_Point:=Position[22];
			TM_MovCmd_Speed:=Proj_Rob_Speed;
			TM_MovCmd_AccelTime:=200;
			TM_MovCmd_Blending:=0;
			TM_MovCmd_PrecisePos:=1;
			TM_MovCmd_RobotPose:='';
			IF VarIO[22] = '' THEN
			TM_MovCmd_Command:='var_switch=10'; //10 = pass; 20 = start stitching; 30 = stop stithing; 40 = gripper on; 50 = gripper off
			ELSE TM_MovCmd_Command:=VarIO[22];
			END_IF;
			TM_MovCmd_ActivateExit:=TRUE;
			TM_MovCmd_CommandID:=1;
			TM_MovCmd_Execute:=FALSE;
			TM_MovCmd_ListenNode:='Listen1';
		
			IF (NOT TM_MovCmd_Done) AND (NOT TM_MovCmd_Error) THEN
				Stage:=222;
			END_IF;
		222:
			TM_MovCmd_Execute:=TRUE;
			IF TM_MovCmd_Done AND Index_STR > 22 THEN
				Stage:=230;
			ELSIF TM_MovCmd_Error THEN
				Stage:=9999;
			END_IF;	
		230:
			TM_MovCmd_Enable:=FALSE;
			MovementIndicatorStage:=Stage;
			IF (NOT TM_MovCmd_Done) AND (NOT TM_MovCmd_Error) AND (NOT TM_MovCmd_Busy) THEN
				Stage:=231;
			END_IF;	
		
		231:
			StepMove:=23;
			TM_MovCmd_Enable:=TRUE;
			TM_MovCmd_Movement:=MovType[23];
			IF MovType[23] = 'PTP'  THEN
			TM_MovCmd_DataFormat:='CPP';
			ELSE TM_MovCmd_DataFormat:='CPR';
			END_IF;
			TM_MovCmd_Point:=Position[23];
			TM_MovCmd_Speed:=Proj_Rob_Speed;
			TM_MovCmd_AccelTime:=200;
			TM_MovCmd_Blending:=0;
			TM_MovCmd_PrecisePos:=1;
			TM_MovCmd_RobotPose:='';
			IF VarIO[23] = '' THEN
			TM_MovCmd_Command:='var_switch=10'; //10 = pass; 20 = start stitching; 30 = stop stithing; 40 = gripper on; 50 = gripper off
			ELSE TM_MovCmd_Command:=VarIO[23];
			END_IF;
			TM_MovCmd_ActivateExit:=TRUE;
			TM_MovCmd_CommandID:=1;
			TM_MovCmd_Execute:=FALSE;
			TM_MovCmd_ListenNode:='Listen1';
		
			IF (NOT TM_MovCmd_Done) AND (NOT TM_MovCmd_Error) THEN
				Stage:=232;
			END_IF;
		232:
			TM_MovCmd_Execute:=TRUE;
			IF TM_MovCmd_Done AND Index_STR > 23 THEN
				Stage:=240;
			ELSIF TM_MovCmd_Error THEN
				Stage:=9999;
			END_IF;	
		240:
			TM_MovCmd_Enable:=FALSE;
			MovementIndicatorStage:=Stage;
			IF (NOT TM_MovCmd_Done) AND (NOT TM_MovCmd_Error) AND (NOT TM_MovCmd_Busy) THEN
				Stage:=241;
			END_IF;	
		
		241:
			StepMove:=24;
			TM_MovCmd_Enable:=TRUE;
			TM_MovCmd_Movement:=MovType[24];
			IF MovType[24] = 'PTP'  THEN
			TM_MovCmd_DataFormat:='CPP';
			ELSE TM_MovCmd_DataFormat:='CPR';
			END_IF;
			TM_MovCmd_Point:=Position[24];
			TM_MovCmd_Speed:=Proj_Rob_Speed;
			TM_MovCmd_AccelTime:=200;
			TM_MovCmd_Blending:=0;
			TM_MovCmd_PrecisePos:=1;
			TM_MovCmd_RobotPose:='';
			IF VarIO[24] = '' THEN
			TM_MovCmd_Command:='var_switch=10'; //10 = pass; 20 = start stitching; 30 = stop stithing; 40 = gripper on; 50 = gripper off
			ELSE TM_MovCmd_Command:=VarIO[24];
			END_IF;
			TM_MovCmd_ActivateExit:=TRUE;
			TM_MovCmd_CommandID:=1;
			TM_MovCmd_Execute:=FALSE;
			TM_MovCmd_ListenNode:='Listen1';
		
			IF (NOT TM_MovCmd_Done) AND (NOT TM_MovCmd_Error) THEN
				Stage:=242;
			END_IF;
		242:
			TM_MovCmd_Execute:=TRUE;
			IF TM_MovCmd_Done AND Index_STR > 24 THEN
				Stage:=250;
			ELSIF TM_MovCmd_Error THEN
				Stage:=9999;
			END_IF;				
		250:
			TM_MovCmd_Enable:=FALSE;
			MovementIndicatorStage:=Stage;
			IF (NOT TM_MovCmd_Done) AND (NOT TM_MovCmd_Error) AND (NOT TM_MovCmd_Busy) THEN
				Stage:=251;
			END_IF;	
		
		251:
			StepMove:=25;
			TM_MovCmd_Enable:=TRUE;
			TM_MovCmd_Movement:=MovType[25];
			IF MovType[25] = 'PTP'  THEN
			TM_MovCmd_DataFormat:='CPP';
			ELSE TM_MovCmd_DataFormat:='CPR';
			END_IF;
			TM_MovCmd_Point:=Position[25];
			TM_MovCmd_Speed:=Proj_Rob_Speed;
			TM_MovCmd_AccelTime:=200;
			TM_MovCmd_Blending:=0;
			TM_MovCmd_PrecisePos:=1;
			TM_MovCmd_RobotPose:='';
			IF VarIO[25] = '' THEN
			TM_MovCmd_Command:='var_switch=10'; //10 = pass; 20 = start stitching; 30 = stop stithing; 40 = gripper on; 50 = gripper off
			ELSE TM_MovCmd_Command:=VarIO[25];
			END_IF;
			TM_MovCmd_ActivateExit:=TRUE;
			TM_MovCmd_CommandID:=1;
			TM_MovCmd_Execute:=FALSE;
			TM_MovCmd_ListenNode:='Listen1';
		
			IF (NOT TM_MovCmd_Done) AND (NOT TM_MovCmd_Error) THEN
				Stage:=252;
			END_IF;
		252:
			TM_MovCmd_Execute:=TRUE;
			IF TM_MovCmd_Done AND Index_STR > 25 THEN
				Stage:=260;
			ELSIF TM_MovCmd_Error THEN
				Stage:=9999;
			END_IF;				
		260:
			TM_MovCmd_Enable:=FALSE;
			MovementIndicatorStage:=Stage;
			IF (NOT TM_MovCmd_Done) AND (NOT TM_MovCmd_Error) AND (NOT TM_MovCmd_Busy) THEN
				Stage:=261;
			END_IF;	
		
		261:
			StepMove:=26;
			TM_MovCmd_Enable:=TRUE;
			TM_MovCmd_Movement:=MovType[26];
			IF MovType[26] = 'PTP'  THEN
			TM_MovCmd_DataFormat:='CPP';
			ELSE TM_MovCmd_DataFormat:='CPR';
			END_IF;
			TM_MovCmd_Point:=Position[26];
			TM_MovCmd_Speed:=Proj_Rob_Speed;
			TM_MovCmd_AccelTime:=200;
			TM_MovCmd_Blending:=0;
			TM_MovCmd_PrecisePos:=1;
			TM_MovCmd_RobotPose:='';
			IF VarIO[26] = '' THEN
			TM_MovCmd_Command:='var_switch=10'; //10 = pass; 20 = start stitching; 30 = stop stithing; 40 = gripper on; 50 = gripper off
			ELSE TM_MovCmd_Command:=VarIO[26];
			END_IF;
			TM_MovCmd_ActivateExit:=TRUE;
			TM_MovCmd_CommandID:=1;
			TM_MovCmd_Execute:=FALSE;
			TM_MovCmd_ListenNode:='Listen1';
		
			IF (NOT TM_MovCmd_Done) AND (NOT TM_MovCmd_Error) THEN
				Stage:=262;
			END_IF;
		262:
			TM_MovCmd_Execute:=TRUE;
			IF TM_MovCmd_Done AND Index_STR > 26 THEN
				Stage:=270;
			ELSIF TM_MovCmd_Error THEN
				Stage:=9999;
			END_IF;		
		270:
			TM_MovCmd_Enable:=FALSE;
			MovementIndicatorStage:=Stage;
			IF (NOT TM_MovCmd_Done) AND (NOT TM_MovCmd_Error) AND (NOT TM_MovCmd_Busy) THEN
				Stage:=271;
			END_IF;	
		
		271:
			StepMove:=27;
			TM_MovCmd_Enable:=TRUE;
			TM_MovCmd_Movement:=MovType[27];
			IF MovType[27] = 'PTP'  THEN
			TM_MovCmd_DataFormat:='CPP';
			ELSE TM_MovCmd_DataFormat:='CPR';
			END_IF;
			TM_MovCmd_Point:=Position[27];
			TM_MovCmd_Speed:=Proj_Rob_Speed;
			TM_MovCmd_AccelTime:=200;
			TM_MovCmd_Blending:=0;
			TM_MovCmd_PrecisePos:=1;
			TM_MovCmd_RobotPose:='';
			IF VarIO[27] = '' THEN
			TM_MovCmd_Command:='var_switch=10'; //10 = pass; 20 = start stitching; 30 = stop stithing; 40 = gripper on; 50 = gripper off
			ELSE TM_MovCmd_Command:=VarIO[27];
			END_IF;
			TM_MovCmd_ActivateExit:=TRUE;
			TM_MovCmd_CommandID:=1;
			TM_MovCmd_Execute:=FALSE;
			TM_MovCmd_ListenNode:='Listen1';
		
			IF (NOT TM_MovCmd_Done) AND (NOT TM_MovCmd_Error) THEN
				Stage:=272;
			END_IF;
		272:
			TM_MovCmd_Execute:=TRUE;
			IF TM_MovCmd_Done AND Index_STR > 27 THEN
				Stage:=280;
			ELSIF TM_MovCmd_Error THEN
				Stage:=9999;
			END_IF;			
		280:
			TM_MovCmd_Enable:=FALSE;
			MovementIndicatorStage:=Stage;
			IF (NOT TM_MovCmd_Done) AND (NOT TM_MovCmd_Error) AND (NOT TM_MovCmd_Busy) THEN
				Stage:=281;
			END_IF;	
		
		281:
			StepMove:=28;
			TM_MovCmd_Enable:=TRUE;
			TM_MovCmd_Movement:=MovType[28];
			IF MovType[28] = 'PTP'  THEN
			TM_MovCmd_DataFormat:='CPP';
			ELSE TM_MovCmd_DataFormat:='CPR';
			END_IF;
			TM_MovCmd_Point:=Position[28];
			TM_MovCmd_Speed:=Proj_Rob_Speed;
			TM_MovCmd_AccelTime:=200;
			TM_MovCmd_Blending:=0;
			TM_MovCmd_PrecisePos:=1;
			TM_MovCmd_RobotPose:='';
			IF VarIO[28] = '' THEN
			TM_MovCmd_Command:='var_switch=10'; //10 = pass; 20 = start stitching; 30 = stop stithing; 40 = gripper on; 50 = gripper off
			ELSE TM_MovCmd_Command:=VarIO[28];
			END_IF;
			TM_MovCmd_ActivateExit:=TRUE;
			TM_MovCmd_CommandID:=1;
			TM_MovCmd_Execute:=FALSE;
			TM_MovCmd_ListenNode:='Listen1';
		
			IF (NOT TM_MovCmd_Done) AND (NOT TM_MovCmd_Error) THEN
				Stage:=282;
			END_IF;
		282:
			TM_MovCmd_Execute:=TRUE;
			IF TM_MovCmd_Done AND Index_STR > 28 THEN
				Stage:=290;
			ELSIF TM_MovCmd_Error THEN
				Stage:=9999;
			END_IF;	
		290:
			TM_MovCmd_Enable:=FALSE;
			MovementIndicatorStage:=Stage;
			IF (NOT TM_MovCmd_Done) AND (NOT TM_MovCmd_Error) AND (NOT TM_MovCmd_Busy) THEN
				Stage:=291;
			END_IF;	
		
		291:
			StepMove:=29;
			TM_MovCmd_Enable:=TRUE;
			TM_MovCmd_Movement:=MovType[29];
			IF MovType[29] = 'PTP'  THEN
			TM_MovCmd_DataFormat:='CPP';
			ELSE TM_MovCmd_DataFormat:='CPR';
			END_IF;
			TM_MovCmd_Point:=Position[29];
			TM_MovCmd_Speed:=Proj_Rob_Speed;
			TM_MovCmd_AccelTime:=200;
			TM_MovCmd_Blending:=0;
			TM_MovCmd_PrecisePos:=1;
			TM_MovCmd_RobotPose:='';
			IF VarIO[29] = '' THEN
			TM_MovCmd_Command:='var_switch=10'; //10 = pass; 20 = start stitching; 30 = stop stithing; 40 = gripper on; 50 = gripper off
			ELSE TM_MovCmd_Command:=VarIO[29];
			END_IF;
			TM_MovCmd_ActivateExit:=TRUE;
			TM_MovCmd_CommandID:=1;
			TM_MovCmd_Execute:=FALSE;
			TM_MovCmd_ListenNode:='Listen1';
		
			IF (NOT TM_MovCmd_Done) AND (NOT TM_MovCmd_Error) THEN
				Stage:=292;
			END_IF;
		292:
			TM_MovCmd_Execute:=TRUE;
			IF TM_MovCmd_Done AND Index_STR > 29 THEN
				Stage:=300;
			ELSIF TM_MovCmd_Error THEN
				Stage:=9999;
			END_IF;				
		300:
			TM_MovCmd_Enable:=FALSE;
			MovementIndicatorStage:=Stage;
			IF (NOT TM_MovCmd_Done) AND (NOT TM_MovCmd_Error) AND (NOT TM_MovCmd_Busy) THEN
				Stage:=301;
			END_IF;	
		
		301:
			StepMove:=30;
			TM_MovCmd_Enable:=TRUE;
			TM_MovCmd_Movement:=MovType[30];
			IF MovType[30] = 'PTP'  THEN
			TM_MovCmd_DataFormat:='CPP';
			ELSE TM_MovCmd_DataFormat:='CPR';
			END_IF;
			TM_MovCmd_Point:=Position[30];
			TM_MovCmd_Speed:=Proj_Rob_Speed;
			TM_MovCmd_AccelTime:=200;
			TM_MovCmd_Blending:=0;
			TM_MovCmd_PrecisePos:=1;
			TM_MovCmd_RobotPose:='';
			IF VarIO[30] = '' THEN
			TM_MovCmd_Command:='var_switch=10'; //10 = pass; 20 = start stitching; 30 = stop stithing; 40 = gripper on; 50 = gripper off
			ELSE TM_MovCmd_Command:=VarIO[30];
			END_IF;
			TM_MovCmd_ActivateExit:=TRUE;
			TM_MovCmd_CommandID:=1;
			TM_MovCmd_Execute:=FALSE;
			TM_MovCmd_ListenNode:='Listen1';
		
			IF (NOT TM_MovCmd_Done) AND (NOT TM_MovCmd_Error) THEN
				Stage:=302;
			END_IF;
		302:
			TM_MovCmd_Execute:=TRUE;
			IF TM_MovCmd_Done AND Index_STR > 30 THEN
				Stage:=310;
			ELSIF TM_MovCmd_Error THEN
				Stage:=9999;
			END_IF;		
		310:
			TM_MovCmd_Enable:=FALSE;
			MovementIndicatorStage:=Stage;
			IF (NOT TM_MovCmd_Done) AND (NOT TM_MovCmd_Error) AND (NOT TM_MovCmd_Busy) THEN
				Stage:=311;
			END_IF;	
		
		311:
		    StepMove:=31;
			TM_MovCmd_Enable:=TRUE;
			TM_MovCmd_Movement:=MovType[31];
			IF MovType[31] = 'PTP'  THEN
			TM_MovCmd_DataFormat:='CPP';
			ELSE TM_MovCmd_DataFormat:='CPR';
			END_IF;
			TM_MovCmd_Point:=Position[31];
			TM_MovCmd_Speed:=Proj_Rob_Speed;
			TM_MovCmd_AccelTime:=200;
			TM_MovCmd_Blending:=0;
			TM_MovCmd_PrecisePos:=1;
			TM_MovCmd_RobotPose:='';
			IF VarIO[31] = '' THEN
			TM_MovCmd_Command:='var_switch=10'; //10 = pass; 20 = start stitching; 30 = stop stithing; 40 = gripper on; 50 = gripper off
			ELSE TM_MovCmd_Command:=VarIO[31];
			END_IF;
			TM_MovCmd_ActivateExit:=TRUE;
			TM_MovCmd_CommandID:=1;
			TM_MovCmd_Execute:=FALSE;
			TM_MovCmd_ListenNode:='Listen1';
		
			IF (NOT TM_MovCmd_Done) AND (NOT TM_MovCmd_Error) THEN
				Stage:=312;
			END_IF;
		312:
			TM_MovCmd_Execute:=TRUE;
			IF TM_MovCmd_Done AND Index_STR > 31 THEN
				Stage:=320;
			ELSIF TM_MovCmd_Error THEN
				Stage:=9999;
			END_IF;		
		320:
			TM_MovCmd_Enable:=FALSE;
			MovementIndicatorStage:=Stage;
			IF (NOT TM_MovCmd_Done) AND (NOT TM_MovCmd_Error) AND (NOT TM_MovCmd_Busy) THEN
				Stage:=321;
			END_IF;	
		
		321:
			StepMove:=32;
			TM_MovCmd_Enable:=TRUE;
			TM_MovCmd_Movement:=MovType[32];
			IF MovType[32] = 'PTP'  THEN
			TM_MovCmd_DataFormat:='CPP';
			ELSE TM_MovCmd_DataFormat:='CPR';
			END_IF;
			TM_MovCmd_Point:=Position[32];
			TM_MovCmd_Speed:=Proj_Rob_Speed;
			TM_MovCmd_AccelTime:=200;
			TM_MovCmd_Blending:=0;
			TM_MovCmd_PrecisePos:=1;
			TM_MovCmd_RobotPose:='';
			IF VarIO[32] = '' THEN
			TM_MovCmd_Command:='var_switch=10'; //10 = pass; 20 = start stitching; 30 = stop stithing; 40 = gripper on; 50 = gripper off
			ELSE TM_MovCmd_Command:=VarIO[32];
			END_IF;
			TM_MovCmd_ActivateExit:=TRUE;
			TM_MovCmd_CommandID:=1;
			TM_MovCmd_Execute:=FALSE;
			TM_MovCmd_ListenNode:='Listen1';
		
			IF (NOT TM_MovCmd_Done) AND (NOT TM_MovCmd_Error) THEN
				Stage:=322;
			END_IF;
		322:
			TM_MovCmd_Execute:=TRUE;
			IF TM_MovCmd_Done AND Index_STR > 32 THEN
				Stage:=330;
			ELSIF TM_MovCmd_Error THEN
				Stage:=9999;
			END_IF;	
		330:
			TM_MovCmd_Enable:=FALSE;
			MovementIndicatorStage:=Stage;
			IF (NOT TM_MovCmd_Done) AND (NOT TM_MovCmd_Error) AND (NOT TM_MovCmd_Busy) THEN
				Stage:=331;
			END_IF;	
		
		331:
			StepMove:=33;
			TM_MovCmd_Enable:=TRUE;
			TM_MovCmd_Movement:=MovType[33];
			IF MovType[33] = 'PTP'  THEN
			TM_MovCmd_DataFormat:='CPP';
			ELSE TM_MovCmd_DataFormat:='CPR';
			END_IF;
			TM_MovCmd_Point:=Position[33];
			TM_MovCmd_Speed:=Proj_Rob_Speed;
			TM_MovCmd_AccelTime:=200;
			TM_MovCmd_Blending:=0;
			TM_MovCmd_PrecisePos:=1;
			TM_MovCmd_RobotPose:='';
			IF VarIO[33] = '' THEN
			TM_MovCmd_Command:='var_switch=10'; //10 = pass; 20 = start stitching; 30 = stop stithing; 40 = gripper on; 50 = gripper off
			ELSE TM_MovCmd_Command:=VarIO[33];
			END_IF;
			TM_MovCmd_ActivateExit:=TRUE;
			TM_MovCmd_CommandID:=1;
			TM_MovCmd_Execute:=FALSE;
			TM_MovCmd_ListenNode:='Listen1';
		
			IF (NOT TM_MovCmd_Done) AND (NOT TM_MovCmd_Error) THEN
				Stage:=332;
			END_IF;
		332:
			TM_MovCmd_Execute:=TRUE;
			IF TM_MovCmd_Done AND Index_STR > 33 THEN
				Stage:=340;
			ELSIF TM_MovCmd_Error THEN
				Stage:=9999;
			END_IF;	
		340:
			TM_MovCmd_Enable:=FALSE;
			MovementIndicatorStage:=Stage;
			IF (NOT TM_MovCmd_Done) AND (NOT TM_MovCmd_Error) AND (NOT TM_MovCmd_Busy) THEN
				Stage:=341;
			END_IF;	
		
		341:
			StepMove:=34;
			TM_MovCmd_Enable:=TRUE;
			TM_MovCmd_Movement:=MovType[34];
			IF MovType[34] = 'PTP'  THEN
			TM_MovCmd_DataFormat:='CPP';
			ELSE TM_MovCmd_DataFormat:='CPR';
			END_IF;
			TM_MovCmd_Point:=Position[34];
			TM_MovCmd_Speed:=Proj_Rob_Speed;
			TM_MovCmd_AccelTime:=200;
			TM_MovCmd_Blending:=0;
			TM_MovCmd_PrecisePos:=1;
			TM_MovCmd_RobotPose:='';
			IF VarIO[34] = '' THEN
			TM_MovCmd_Command:='var_switch=10'; //10 = pass; 20 = start stitching; 30 = stop stithing; 40 = gripper on; 50 = gripper off
			ELSE TM_MovCmd_Command:=VarIO[34];
			END_IF;
			TM_MovCmd_ActivateExit:=TRUE;
			TM_MovCmd_CommandID:=1;
			TM_MovCmd_Execute:=FALSE;
			TM_MovCmd_ListenNode:='Listen1';
		
			IF (NOT TM_MovCmd_Done) AND (NOT TM_MovCmd_Error) THEN
				Stage:=342;
			END_IF;
		342:
			TM_MovCmd_Execute:=TRUE;
			IF TM_MovCmd_Done AND Index_STR > 34 THEN
				Stage:=350;
			ELSIF TM_MovCmd_Error THEN
				Stage:=9999;
			END_IF;				
		350:
			TM_MovCmd_Enable:=FALSE;
			MovementIndicatorStage:=Stage;
			IF (NOT TM_MovCmd_Done) AND (NOT TM_MovCmd_Error) AND (NOT TM_MovCmd_Busy) THEN
				Stage:=351;
			END_IF;	
		
		351:
			StepMove:=35;
			TM_MovCmd_Enable:=TRUE;
			TM_MovCmd_Movement:=MovType[35];
			IF MovType[35] = 'PTP'  THEN
			TM_MovCmd_DataFormat:='CPP';
			ELSE TM_MovCmd_DataFormat:='CPR';
			END_IF;
			TM_MovCmd_Point:=Position[35];
			TM_MovCmd_Speed:=Proj_Rob_Speed;
			TM_MovCmd_AccelTime:=200;
			TM_MovCmd_Blending:=0;
			TM_MovCmd_PrecisePos:=1;
			TM_MovCmd_RobotPose:='';
			IF VarIO[35] = '' THEN
			TM_MovCmd_Command:='var_switch=10'; //10 = pass; 20 = start stitching; 30 = stop stithing; 40 = gripper on; 50 = gripper off
			ELSE TM_MovCmd_Command:=VarIO[35];
			END_IF;
			TM_MovCmd_ActivateExit:=TRUE;
			TM_MovCmd_CommandID:=1;
			TM_MovCmd_Execute:=FALSE;
			TM_MovCmd_ListenNode:='Listen1';
		
			IF (NOT TM_MovCmd_Done) AND (NOT TM_MovCmd_Error) THEN
				Stage:=352;
			END_IF;
		352:
			TM_MovCmd_Execute:=TRUE;
			IF TM_MovCmd_Done AND Index_STR > 35 THEN
				Stage:=360;
			ELSIF TM_MovCmd_Error THEN
				Stage:=9999;
			END_IF;				
		360:
			TM_MovCmd_Enable:=FALSE;
			MovementIndicatorStage:=Stage;
			IF (NOT TM_MovCmd_Done) AND (NOT TM_MovCmd_Error) AND (NOT TM_MovCmd_Busy) THEN
				Stage:=361;
			END_IF;	
		
		361:
			StepMove:=36;
			TM_MovCmd_Enable:=TRUE;
			TM_MovCmd_Movement:=MovType[36];
			IF MovType[36] = 'PTP'  THEN
			TM_MovCmd_DataFormat:='CPP';
			ELSE TM_MovCmd_DataFormat:='CPR';
			END_IF;
			TM_MovCmd_Point:=Position[36];
			TM_MovCmd_Speed:=Proj_Rob_Speed;
			TM_MovCmd_AccelTime:=200;
			TM_MovCmd_Blending:=0;
			TM_MovCmd_PrecisePos:=1;
			TM_MovCmd_RobotPose:='';
			IF VarIO[36] = '' THEN
			TM_MovCmd_Command:='var_switch=10'; //10 = pass; 20 = start stitching; 30 = stop stithing; 40 = gripper on; 50 = gripper off
			ELSE TM_MovCmd_Command:=VarIO[36];
			END_IF;
			TM_MovCmd_ActivateExit:=TRUE;
			TM_MovCmd_CommandID:=1;
			TM_MovCmd_Execute:=FALSE;
			TM_MovCmd_ListenNode:='Listen1';
		
			IF (NOT TM_MovCmd_Done) AND (NOT TM_MovCmd_Error) THEN
				Stage:=362;
			END_IF;
		362:
			TM_MovCmd_Execute:=TRUE;
			IF TM_MovCmd_Done AND Index_STR > 36 THEN
				Stage:=370;
			ELSIF TM_MovCmd_Error THEN
				Stage:=9999;
			END_IF;		
		370:
			TM_MovCmd_Enable:=FALSE;
			MovementIndicatorStage:=Stage;
			IF (NOT TM_MovCmd_Done) AND (NOT TM_MovCmd_Error) AND (NOT TM_MovCmd_Busy) THEN
				Stage:=371;
			END_IF;	
		
		371:
			StepMove:=37;
			TM_MovCmd_Enable:=TRUE;
			TM_MovCmd_Movement:=MovType[37];
			IF MovType[37] = 'PTP'  THEN
			TM_MovCmd_DataFormat:='CPP';
			ELSE TM_MovCmd_DataFormat:='CPR';
			END_IF;
			TM_MovCmd_Point:=Position[37];
			TM_MovCmd_Speed:=Proj_Rob_Speed;
			TM_MovCmd_AccelTime:=200;
			TM_MovCmd_Blending:=0;
			TM_MovCmd_PrecisePos:=1;
			TM_MovCmd_RobotPose:='';
			IF VarIO[37] = '' THEN
			TM_MovCmd_Command:='var_switch=10'; //10 = pass; 20 = start stitching; 30 = stop stithing; 40 = gripper on; 50 = gripper off
			ELSE TM_MovCmd_Command:=VarIO[37];
			END_IF;
			TM_MovCmd_ActivateExit:=TRUE;
			TM_MovCmd_CommandID:=1;
			TM_MovCmd_Execute:=FALSE;
			TM_MovCmd_ListenNode:='Listen1';
		
			IF (NOT TM_MovCmd_Done) AND (NOT TM_MovCmd_Error) THEN
				Stage:=372;
			END_IF;
		372:
			TM_MovCmd_Execute:=TRUE;
			IF TM_MovCmd_Done AND Index_STR > 37 THEN
				Stage:=380;
			ELSIF TM_MovCmd_Error THEN
				Stage:=9999;
			END_IF;			
		380:
			TM_MovCmd_Enable:=FALSE;
			MovementIndicatorStage:=Stage;
			IF (NOT TM_MovCmd_Done) AND (NOT TM_MovCmd_Error) AND (NOT TM_MovCmd_Busy) THEN
				Stage:=381;
			END_IF;	
		
		381:
			StepMove:=38;
			TM_MovCmd_Enable:=TRUE;
			TM_MovCmd_Movement:=MovType[38];
			IF MovType[38] = 'PTP'  THEN
			TM_MovCmd_DataFormat:='CPP';
			ELSE TM_MovCmd_DataFormat:='CPR';
			END_IF;
			TM_MovCmd_Point:=Position[38];
			TM_MovCmd_Speed:=Proj_Rob_Speed;
			TM_MovCmd_AccelTime:=200;
			TM_MovCmd_Blending:=0;
			TM_MovCmd_PrecisePos:=1;
			TM_MovCmd_RobotPose:='';
			IF VarIO[38] = '' THEN
			TM_MovCmd_Command:='var_switch=10'; //10 = pass; 20 = start stitching; 30 = stop stithing; 40 = gripper on; 50 = gripper off
			ELSE TM_MovCmd_Command:=VarIO[38];
			END_IF;
			TM_MovCmd_ActivateExit:=TRUE;
			TM_MovCmd_CommandID:=1;
			TM_MovCmd_Execute:=FALSE;
			TM_MovCmd_ListenNode:='Listen1';
		
			IF (NOT TM_MovCmd_Done) AND (NOT TM_MovCmd_Error) THEN
				Stage:=382;
			END_IF;
		382:
			TM_MovCmd_Execute:=TRUE;
			IF TM_MovCmd_Done AND Index_STR > 38 THEN
				Stage:=390;
			ELSIF TM_MovCmd_Error THEN
				Stage:=9999;
			END_IF;	
		390:
			TM_MovCmd_Enable:=FALSE;
			MovementIndicatorStage:=Stage;
			IF (NOT TM_MovCmd_Done) AND (NOT TM_MovCmd_Error) AND (NOT TM_MovCmd_Busy) THEN
				Stage:=391;
			END_IF;	
		
		391:
			StepMove:=39;
			TM_MovCmd_Enable:=TRUE;
			TM_MovCmd_Movement:=MovType[39];
			IF MovType[39] = 'PTP'  THEN
			TM_MovCmd_DataFormat:='CPP';
			ELSE TM_MovCmd_DataFormat:='CPR';
			END_IF;
			TM_MovCmd_Point:=Position[39];
			TM_MovCmd_Speed:=Proj_Rob_Speed;
			TM_MovCmd_AccelTime:=200;
			TM_MovCmd_Blending:=0;
			TM_MovCmd_PrecisePos:=1;
			TM_MovCmd_RobotPose:='';
			IF VarIO[39] = '' THEN
			TM_MovCmd_Command:='var_switch=10'; //10 = pass; 20 = start stitching; 30 = stop stithing; 40 = gripper on; 50 = gripper off
			ELSE TM_MovCmd_Command:=VarIO[39];
			END_IF;
			TM_MovCmd_ActivateExit:=TRUE;
			TM_MovCmd_CommandID:=1;
			TM_MovCmd_Execute:=FALSE;
			TM_MovCmd_ListenNode:='Listen1';
		
			IF (NOT TM_MovCmd_Done) AND (NOT TM_MovCmd_Error) THEN
				Stage:=392;
			END_IF;
		392:
			TM_MovCmd_Execute:=TRUE;
			IF TM_MovCmd_Done AND Index_STR > 39 THEN
				Stage:=400;
			ELSIF TM_MovCmd_Error THEN
				Stage:=9999;
			END_IF;	
		400:
			TM_MovCmd_Enable:=FALSE;
			MovementIndicatorStage:=Stage;
			IF (NOT TM_MovCmd_Done) AND (NOT TM_MovCmd_Error) AND (NOT TM_MovCmd_Busy) THEN
				Stage:=401;
			END_IF;	
		
		401:
			StepMove:=40;
			TM_MovCmd_Enable:=TRUE;
			TM_MovCmd_Movement:=MovType[40];
			IF MovType[40] = 'PTP'  THEN
			TM_MovCmd_DataFormat:='CPP';
			ELSE TM_MovCmd_DataFormat:='CPR';
			END_IF;
			TM_MovCmd_Point:=Position[40];
			TM_MovCmd_Speed:=Proj_Rob_Speed;
			TM_MovCmd_AccelTime:=200;
			TM_MovCmd_Blending:=0;
			TM_MovCmd_PrecisePos:=1;
			TM_MovCmd_RobotPose:='';
			IF VarIO[40] = '' THEN
			TM_MovCmd_Command:='var_switch=10'; //10 = pass; 20 = start stitching; 30 = stop stithing; 40 = gripper on; 50 = gripper off
			ELSE TM_MovCmd_Command:=VarIO[40];
			END_IF;
			TM_MovCmd_ActivateExit:=TRUE;
			TM_MovCmd_CommandID:=1;
			TM_MovCmd_Execute:=FALSE;
			TM_MovCmd_ListenNode:='Listen1';
		
			IF (NOT TM_MovCmd_Done) AND (NOT TM_MovCmd_Error) THEN
				Stage:=402;
			END_IF;
		402:
			TM_MovCmd_Execute:=TRUE;
			IF TM_MovCmd_Done AND Index_STR > 40 THEN
				Stage:=410;
			ELSIF TM_MovCmd_Error THEN
				Stage:=9999;
			END_IF;		
		410:
			TM_MovCmd_Enable:=FALSE;
			MovementIndicatorStage:=Stage;
			IF (NOT TM_MovCmd_Done) AND (NOT TM_MovCmd_Error) AND (NOT TM_MovCmd_Busy) THEN
				Stage:=411;
			END_IF;	
		
		411:
			StepMove:=41;
			TM_MovCmd_Enable:=TRUE;
			TM_MovCmd_Movement:=MovType[41];
			IF MovType[41] = 'PTP'  THEN
			TM_MovCmd_DataFormat:='CPP';
			ELSE TM_MovCmd_DataFormat:='CPR';
			END_IF;
			TM_MovCmd_Point:=Position[41];
			TM_MovCmd_Speed:=Proj_Rob_Speed;
			TM_MovCmd_AccelTime:=200;
			TM_MovCmd_Blending:=0;
			TM_MovCmd_PrecisePos:=1;
			TM_MovCmd_RobotPose:='';
			IF VarIO[41] = '' THEN
			TM_MovCmd_Command:='var_switch=10'; //10 = pass; 20 = start stitching; 30 = stop stithing; 40 = gripper on; 50 = gripper off
			ELSE TM_MovCmd_Command:=VarIO[41];
			END_IF;
			TM_MovCmd_ActivateExit:=TRUE;
			TM_MovCmd_CommandID:=1;
			TM_MovCmd_Execute:=FALSE;
			TM_MovCmd_ListenNode:='Listen1';
		
			IF (NOT TM_MovCmd_Done) AND (NOT TM_MovCmd_Error) THEN
				Stage:=412;
			END_IF;
		412:
			TM_MovCmd_Execute:=TRUE;
			IF TM_MovCmd_Done AND Index_STR > 41 THEN
				Stage:=420;
			ELSIF TM_MovCmd_Error THEN
				Stage:=9999;
			END_IF;		
		420:
			TM_MovCmd_Enable:=FALSE;
			MovementIndicatorStage:=Stage;
			IF (NOT TM_MovCmd_Done) AND (NOT TM_MovCmd_Error) AND (NOT TM_MovCmd_Busy) THEN
				Stage:=421;
			END_IF;	
		
		421:
			StepMove:=42;
			TM_MovCmd_Enable:=TRUE;
			TM_MovCmd_Movement:=MovType[42];
			IF MovType[42] = 'PTP'  THEN
			TM_MovCmd_DataFormat:='CPP';
			ELSE TM_MovCmd_DataFormat:='CPR';
			END_IF;
			TM_MovCmd_Point:=Position[42];
			TM_MovCmd_Speed:=Proj_Rob_Speed;
			TM_MovCmd_AccelTime:=200;
			TM_MovCmd_Blending:=0;
			TM_MovCmd_PrecisePos:=1;
			TM_MovCmd_RobotPose:='';
			IF VarIO[42] = '' THEN
			TM_MovCmd_Command:='var_switch=10'; //10 = pass; 20 = start stitching; 30 = stop stithing; 40 = gripper on; 50 = gripper off
			ELSE TM_MovCmd_Command:=VarIO[42];
			END_IF;
			TM_MovCmd_ActivateExit:=TRUE;
			TM_MovCmd_CommandID:=1;
			TM_MovCmd_Execute:=FALSE;
			TM_MovCmd_ListenNode:='Listen1';
		
			IF (NOT TM_MovCmd_Done) AND (NOT TM_MovCmd_Error) THEN
				Stage:=422;
			END_IF;
		422:
			TM_MovCmd_Execute:=TRUE;
			IF TM_MovCmd_Done AND Index_STR > 42 THEN
				Stage:=430;
			ELSIF TM_MovCmd_Error THEN
				Stage:=9999;
			END_IF;	
		430:
			TM_MovCmd_Enable:=FALSE;
			MovementIndicatorStage:=Stage;
			IF (NOT TM_MovCmd_Done) AND (NOT TM_MovCmd_Error) AND (NOT TM_MovCmd_Busy) THEN
				Stage:=441;
			END_IF;	
		
		431:
			StepMove:=43;
			TM_MovCmd_Enable:=TRUE;
			TM_MovCmd_Movement:=MovType[43];
			IF MovType[43] = 'PTP'  THEN
			TM_MovCmd_DataFormat:='CPP';
			ELSE TM_MovCmd_DataFormat:='CPR';
			END_IF;
			TM_MovCmd_Point:=Position[43];
			TM_MovCmd_Speed:=Proj_Rob_Speed;
			TM_MovCmd_AccelTime:=200;
			TM_MovCmd_Blending:=0;
			TM_MovCmd_PrecisePos:=1;
			TM_MovCmd_RobotPose:='';
			IF VarIO[43] = '' THEN
			TM_MovCmd_Command:='var_switch=10'; //10 = pass; 20 = start stitching; 30 = stop stithing; 40 = gripper on; 50 = gripper off
			ELSE TM_MovCmd_Command:=VarIO[43];
			END_IF;
			TM_MovCmd_ActivateExit:=TRUE;
			TM_MovCmd_CommandID:=1;
			TM_MovCmd_Execute:=FALSE;
			TM_MovCmd_ListenNode:='Listen1';
		
			IF (NOT TM_MovCmd_Done) AND (NOT TM_MovCmd_Error) THEN
				Stage:=432;
			END_IF;
		432:
			TM_MovCmd_Execute:=TRUE;
			IF TM_MovCmd_Done AND Index_STR > 43 THEN
				Stage:=440;
			ELSIF TM_MovCmd_Error THEN
				Stage:=9999;
			END_IF;	
		440:
			TM_MovCmd_Enable:=FALSE;
			MovementIndicatorStage:=Stage;
			IF (NOT TM_MovCmd_Done) AND (NOT TM_MovCmd_Error) AND (NOT TM_MovCmd_Busy) THEN
				Stage:=441;
			END_IF;	
		
		441:
			StepMove:=44;
			TM_MovCmd_Enable:=TRUE;
			TM_MovCmd_Movement:=MovType[44];
			IF MovType[44] = 'PTP'  THEN
			TM_MovCmd_DataFormat:='CPP';
			ELSE TM_MovCmd_DataFormat:='CPR';
			END_IF;
			TM_MovCmd_Point:=Position[44];
			TM_MovCmd_Speed:=Proj_Rob_Speed;
			TM_MovCmd_AccelTime:=200;
			TM_MovCmd_Blending:=0;
			TM_MovCmd_PrecisePos:=1;
			TM_MovCmd_RobotPose:='';
			IF VarIO[44] = '' THEN
			TM_MovCmd_Command:='var_switch=10'; //10 = pass; 20 = start stitching; 30 = stop stithing; 40 = gripper on; 50 = gripper off
			ELSE TM_MovCmd_Command:=VarIO[44];
			END_IF;
			TM_MovCmd_ActivateExit:=TRUE;
			TM_MovCmd_CommandID:=1;
			TM_MovCmd_Execute:=FALSE;
			TM_MovCmd_ListenNode:='Listen1';
		
			IF (NOT TM_MovCmd_Done) AND (NOT TM_MovCmd_Error) THEN
				Stage:=442;
			END_IF;
		442:
			TM_MovCmd_Execute:=TRUE;
			IF TM_MovCmd_Done AND Index_STR > 44 THEN
				Stage:=450;
			ELSIF TM_MovCmd_Error THEN
				Stage:=9999;
			END_IF;				
		450:
			TM_MovCmd_Enable:=FALSE;
			MovementIndicatorStage:=Stage;
			IF (NOT TM_MovCmd_Done) AND (NOT TM_MovCmd_Error) AND (NOT TM_MovCmd_Busy) THEN
				Stage:=451;
			END_IF;	
		
		451:
			StepMove:=45;
			TM_MovCmd_Enable:=TRUE;
			TM_MovCmd_Movement:=MovType[45];
			IF MovType[45] = 'PTP'  THEN
			TM_MovCmd_DataFormat:='CPP';
			ELSE TM_MovCmd_DataFormat:='CPR';
			END_IF;
			TM_MovCmd_Point:=Position[45];
			TM_MovCmd_Speed:=Proj_Rob_Speed;
			TM_MovCmd_AccelTime:=200;
			TM_MovCmd_Blending:=0;
			TM_MovCmd_PrecisePos:=1;
			TM_MovCmd_RobotPose:='';
			IF VarIO[45] = '' THEN
			TM_MovCmd_Command:='var_switch=10'; //10 = pass; 20 = start stitching; 30 = stop stithing; 40 = gripper on; 50 = gripper off
			ELSE TM_MovCmd_Command:=VarIO[45];
			END_IF;
			TM_MovCmd_ActivateExit:=TRUE;
			TM_MovCmd_CommandID:=1;
			TM_MovCmd_Execute:=FALSE;
			TM_MovCmd_ListenNode:='Listen1';
		
			IF (NOT TM_MovCmd_Done) AND (NOT TM_MovCmd_Error) THEN
				Stage:=452;
			END_IF;
		452:
			TM_MovCmd_Execute:=TRUE;
			IF TM_MovCmd_Done AND Index_STR > 45 THEN
				Stage:=460;
			ELSIF TM_MovCmd_Error THEN
				Stage:=9999;
			END_IF;				
		460:
			TM_MovCmd_Enable:=FALSE;
			MovementIndicatorStage:=Stage;
			IF (NOT TM_MovCmd_Done) AND (NOT TM_MovCmd_Error) AND (NOT TM_MovCmd_Busy) THEN
				Stage:=461;
			END_IF;	
		
		461:
			StepMove:=46;
			TM_MovCmd_Enable:=TRUE;
			TM_MovCmd_Movement:=MovType[46];
			IF MovType[46] = 'PTP'  THEN
			TM_MovCmd_DataFormat:='CPP';
			ELSE TM_MovCmd_DataFormat:='CPR';
			END_IF;
			TM_MovCmd_Point:=Position[46];
			TM_MovCmd_Speed:=Proj_Rob_Speed;
			TM_MovCmd_AccelTime:=200;
			TM_MovCmd_Blending:=0;
			TM_MovCmd_PrecisePos:=1;
			TM_MovCmd_RobotPose:='';
			IF VarIO[46] = '' THEN
			TM_MovCmd_Command:='var_switch=10'; //10 = pass; 20 = start stitching; 30 = stop stithing; 40 = gripper on; 50 = gripper off
			ELSE TM_MovCmd_Command:=VarIO[46];
			END_IF;
			TM_MovCmd_ActivateExit:=TRUE;
			TM_MovCmd_CommandID:=1;
			TM_MovCmd_Execute:=FALSE;
			TM_MovCmd_ListenNode:='Listen1';
		
			IF (NOT TM_MovCmd_Done) AND (NOT TM_MovCmd_Error) THEN
				Stage:=462;
			END_IF;
		462:
			TM_MovCmd_Execute:=TRUE;
			IF TM_MovCmd_Done AND Index_STR > 46 THEN
				Stage:=470;
			ELSIF TM_MovCmd_Error THEN
				Stage:=9999;
			END_IF;		
		470:
			TM_MovCmd_Enable:=FALSE;
			MovementIndicatorStage:=Stage;
			IF (NOT TM_MovCmd_Done) AND (NOT TM_MovCmd_Error) AND (NOT TM_MovCmd_Busy) THEN
				Stage:=471;
			END_IF;	
		
		471:
			StepMove:=47;
			TM_MovCmd_Enable:=TRUE;
			TM_MovCmd_Movement:=MovType[47];
			IF MovType[47] = 'PTP'  THEN
			TM_MovCmd_DataFormat:='CPP';
			ELSE TM_MovCmd_DataFormat:='CPR';
			END_IF;
			TM_MovCmd_Point:=Position[47];
			TM_MovCmd_Speed:=Proj_Rob_Speed;
			TM_MovCmd_AccelTime:=200;
			TM_MovCmd_Blending:=0;
			TM_MovCmd_PrecisePos:=1;
			TM_MovCmd_RobotPose:='';
			IF VarIO[47] = '' THEN
			TM_MovCmd_Command:='var_switch=10'; //10 = pass; 20 = start stitching; 30 = stop stithing; 40 = gripper on; 50 = gripper off
			ELSE TM_MovCmd_Command:=VarIO[47];
			END_IF;
			TM_MovCmd_ActivateExit:=TRUE;
			TM_MovCmd_CommandID:=1;
			TM_MovCmd_Execute:=FALSE;
			TM_MovCmd_ListenNode:='Listen1';
		
			IF (NOT TM_MovCmd_Done) AND (NOT TM_MovCmd_Error) THEN
				Stage:=472;
			END_IF;
		472:
			TM_MovCmd_Execute:=TRUE;
			IF TM_MovCmd_Done AND Index_STR > 47 THEN
				Stage:=480;
			ELSIF TM_MovCmd_Error THEN
				Stage:=9999;
			END_IF;			
		480:
			TM_MovCmd_Enable:=FALSE;
			MovementIndicatorStage:=Stage;
			IF (NOT TM_MovCmd_Done) AND (NOT TM_MovCmd_Error) AND (NOT TM_MovCmd_Busy) THEN
				Stage:=481;
			END_IF;	
		
		481:
			StepMove:=48;
			TM_MovCmd_Enable:=TRUE;
			TM_MovCmd_Movement:=MovType[48];
			IF MovType[48] = 'PTP'  THEN
			TM_MovCmd_DataFormat:='CPP';
			ELSE TM_MovCmd_DataFormat:='CPR';
			END_IF;
			TM_MovCmd_Point:=Position[48];
			TM_MovCmd_Speed:=Proj_Rob_Speed;
			TM_MovCmd_AccelTime:=200;
			TM_MovCmd_Blending:=0;
			TM_MovCmd_PrecisePos:=1;
			TM_MovCmd_RobotPose:='';
			IF VarIO[48] = '' THEN
			TM_MovCmd_Command:='var_switch=10'; //10 = pass; 20 = start stitching; 30 = stop stithing; 40 = gripper on; 50 = gripper off
			ELSE TM_MovCmd_Command:=VarIO[48];
			END_IF;
			TM_MovCmd_ActivateExit:=TRUE;
			TM_MovCmd_CommandID:=1;
			TM_MovCmd_Execute:=FALSE;
			TM_MovCmd_ListenNode:='Listen1';
		
			IF (NOT TM_MovCmd_Done) AND (NOT TM_MovCmd_Error) THEN
				Stage:=482;
			END_IF;
		482:
			TM_MovCmd_Execute:=TRUE;
			IF TM_MovCmd_Done AND Index_STR > 48 THEN
				Stage:=490;
			ELSIF TM_MovCmd_Error THEN
				Stage:=9999;
			END_IF;	
		490:
			TM_MovCmd_Enable:=FALSE;
			MovementIndicatorStage:=Stage;
			IF (NOT TM_MovCmd_Done) AND (NOT TM_MovCmd_Error) AND (NOT TM_MovCmd_Busy) THEN
				Stage:=491;
			END_IF;	
		
		491:
			StepMove:=49;
			TM_MovCmd_Enable:=TRUE;
			TM_MovCmd_Movement:=MovType[49];
			IF MovType[49] = 'PTP'  THEN
			TM_MovCmd_DataFormat:='CPP';
			ELSE TM_MovCmd_DataFormat:='CPR';
			END_IF;
			TM_MovCmd_Point:=Position[49];
			TM_MovCmd_Speed:=Proj_Rob_Speed;
			TM_MovCmd_AccelTime:=200;
			TM_MovCmd_Blending:=0;
			TM_MovCmd_PrecisePos:=1;
			TM_MovCmd_RobotPose:='';
			IF VarIO[49] = '' THEN
			TM_MovCmd_Command:='var_switch=10'; //10 = pass; 20 = start stitching; 30 = stop stithing; 40 = gripper on; 50 = gripper off
			ELSE TM_MovCmd_Command:=VarIO[49];
			END_IF;
			TM_MovCmd_ActivateExit:=TRUE;
			TM_MovCmd_CommandID:=1;
			TM_MovCmd_Execute:=FALSE;
			TM_MovCmd_ListenNode:='Listen1';
		
			IF (NOT TM_MovCmd_Done) AND (NOT TM_MovCmd_Error) THEN
				Stage:=492;
			END_IF;
		492:
			TM_MovCmd_Execute:=TRUE;
			IF TM_MovCmd_Done AND Index_STR > 49 THEN
				Stage:=500;
			ELSIF TM_MovCmd_Error THEN
				Stage:=9999;
			END_IF;				
		500:
			TM_MovCmd_Enable:=FALSE;
			MovementIndicatorStage:=Stage;
			IF (NOT TM_MovCmd_Done) AND (NOT TM_MovCmd_Error) AND (NOT TM_MovCmd_Busy) THEN
				Stage:=501;
			END_IF;	
		
		501:
			StepMove:=50;
			TM_MovCmd_Enable:=TRUE;
			TM_MovCmd_Movement:=MovType[50];
			IF MovType[50] = 'PTP'  THEN
			TM_MovCmd_DataFormat:='CPP';
			ELSE TM_MovCmd_DataFormat:='CPR';
			END_IF;
			TM_MovCmd_Point:=Position[50];
			TM_MovCmd_Speed:=Proj_Rob_Speed;
			TM_MovCmd_AccelTime:=200;
			TM_MovCmd_Blending:=0;
			TM_MovCmd_PrecisePos:=1;
			TM_MovCmd_RobotPose:='';
			IF VarIO[50] = '' THEN
			TM_MovCmd_Command:='var_switch=10'; //10 = pass; 20 = start stitching; 30 = stop stithing; 40 = gripper on; 50 = gripper off
			ELSE TM_MovCmd_Command:=VarIO[50];
			END_IF;
			TM_MovCmd_ActivateExit:=TRUE;
			TM_MovCmd_CommandID:=1;
			TM_MovCmd_Execute:=FALSE;
			TM_MovCmd_ListenNode:='Listen1';
		
			IF (NOT TM_MovCmd_Done) AND (NOT TM_MovCmd_Error) THEN
				Stage:=502;
			END_IF;
		502:
			TM_MovCmd_Execute:=TRUE;
			IF TM_MovCmd_Done AND Index_STR > 50 THEN
				Stage:=510;
			ELSIF TM_MovCmd_Error THEN
				Stage:=9999;
			END_IF;		
		510:
			TM_MovCmd_Enable:=FALSE;
			MovementIndicatorStage:=Stage;
			IF (NOT TM_MovCmd_Done) AND (NOT TM_MovCmd_Error) AND (NOT TM_MovCmd_Busy) THEN
				Stage:=511;
			END_IF;	
		
		511:
			StepMove:=51;
			TM_MovCmd_Enable:=TRUE;
			TM_MovCmd_Movement:=MovType[51];
			IF MovType[51] = 'PTP'  THEN
			TM_MovCmd_DataFormat:='CPP';
			ELSE TM_MovCmd_DataFormat:='CPR';
			END_IF;
			TM_MovCmd_Point:=Position[51];
			TM_MovCmd_Speed:=Proj_Rob_Speed;
			TM_MovCmd_AccelTime:=200;
			TM_MovCmd_Blending:=0;
			TM_MovCmd_PrecisePos:=1;
			TM_MovCmd_RobotPose:='';
			IF VarIO[51] = '' THEN
			TM_MovCmd_Command:='var_switch=10'; //10 = pass; 20 = start stitching; 30 = stop stithing; 40 = gripper on; 50 = gripper off
			ELSE TM_MovCmd_Command:=VarIO[51];
			END_IF;
			TM_MovCmd_ActivateExit:=TRUE;
			TM_MovCmd_CommandID:=1;
			TM_MovCmd_Execute:=FALSE;
			TM_MovCmd_ListenNode:='Listen1';
		
			IF (NOT TM_MovCmd_Done) AND (NOT TM_MovCmd_Error) THEN
				Stage:=512;
			END_IF;
		512:
			TM_MovCmd_Execute:=TRUE;
			IF TM_MovCmd_Done THEN
				Stage:=9999;
			ELSIF TM_MovCmd_Error THEN
				Stage:=9999;
			END_IF;		

	END_CASE;
	
END_IF;

		//Stitching control based on robot absolute position
		
		IF RobotIO.ControlBox.DO0 = 1 AND Rob_Speed >0 AND StartProgram = 1 THEN 
	  			Run_Stiching:=1;
				Run_Stiching_Man:=0;
				Stitcher_AutoSpeed:=1;
				Speed:=2;
		ELSIF RobotIO.ControlBox.DO0 = 0 AND StartProgram = 1 THEN
				Run_Stiching:=0;
				Run_Stiching_Man:=1;
				Stitcher_AutoSpeed:=0;
			//	IF Relay_Output9 = 0 THEN 
			    Speed:= -2;
			//	END_IF; 
		END_IF;

TM_MovCmd_Instance(
	Done=>TM_MovCmd_Done,
	Busy=>TM_MovCmd_Busy,
	Error=>TM_MovCmd_Error,
	ErrorID=>TM_MovCmd_ErrorID,
	Execute:=TM_MovCmd_Execute,
	RobotID:=ListenNode_Connect_TCP_Socket,
	Movement:=TM_MovCmd_Movement,
	DataFormat:=TM_MovCmd_DataFormat,
	Point:=TM_MovCmd_Point,
	Speed:=TM_MovCmd_Speed,
	AccelTime:=TM_MovCmd_AccelTime,
	Blending:=TM_MovCmd_Blending,
	PrecisePos:=TM_MovCmd_PrecisePos,
	RobotPose:=TM_MovCmd_RobotPose,
	Command:=TM_MovCmd_Command,  
	ActivateExit:=TM_MovCmd_ActivateExit,
	CommandID:=TM_MovCmd_CommandID,
	TimeOut:=T#3600s,
	ListenNode:=TM_MovCmd_ListenNode,
	TimeOutET=>TM_MovCmd_TimeOutET,
	Enable:=TM_MovCmd_Enable
);

TM_ChangeTCP_Instance(
	Enable:=TM_ChangeTCP_Enable,
	Execute:=TM_ChangeTCP_Execute,
	RobotID:=ListenNode_Connect_TCP_Socket,
	TCP:=TM_ChangeTCP_TCP,
	Weight:=TM_ChangeTCP_Weight,
	MomInertia:=TM_ChangeTCP_MomInertia,
	RefFrame:=TM_ChangeTCP_RefFrame,
	Command:=TM_ChangeTCP_Command,
	ActivateExit:=TM_ChangeTCP_ActivateExit,
	ListenNode:=TM_ChangeTCP_ListenNode,
	TimeOut:=T#3600s,
	CommandID:=TM_ChangeTCP_CommandID,
	Done=>TM_ChangeTCP_Done,
	Busy=>TM_ChangeTCP_Busy,
	Error=>TM_ChangeTCP_Error,
	ErrorID=>TM_ChangeTCP_ErrorID,
	TimeOutET=>TM_ChangeTCP_TimeOutET
);

TM_ChangeLoad_Instance(
	Enable:=TM_ChangeLoad_Enable,
	Execute:=TM_ChangeLoad_Execute,
	RobotID:=ListenNode_Connect_TCP_Socket,
	Payload:=TM_ChangeLoad_Payload,
	Command:=TM_ChangeLoad_Command,
	ActivateExit:=TM_ChangeLoad_ActivateExit,
	ListenNode:=TM_ChangeLoad_ListenNode,
	TimeOut:=T#3600s,
	CommandID:=TM_ChangeLoad_CommandID,
	Done=>TM_ChangeLoad_Done,
	Busy=>TM_ChangeLoad_Busy,
	Error=>TM_ChangeLoad_Error,
	ErrorID=>TM_ChangeLoad_ErrorID,
	TimeOutET=>TM_ChangeLoad_TimeOutET
);

